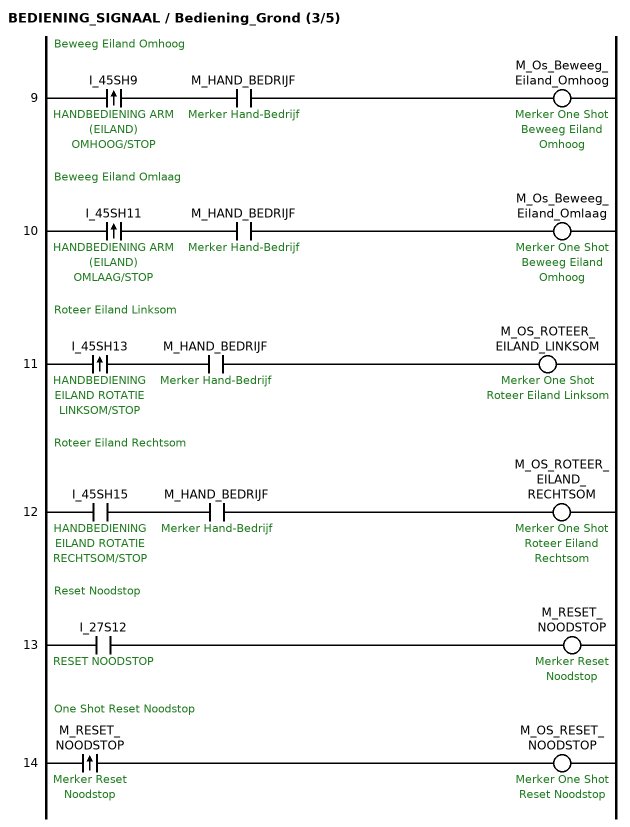
; [picture p96: BEDIENING_SIGNAAL / Bediening_Grond, rungs 9-14]
; rung 9: Beweeg Eiland Omhoog
@LD I_45SH9  ; HANDBEDIENING ARM (EILAND) OMHOOG/STOP
AND M_HAND_BEDRIJF  ; Merker Hand-Bedrijf
OUT M_Os_Beweeg_Eiland_Omhoog  ; Merker One Shot Beweeg Eiland Omhoog
; rung 10: Beweeg Eiland Omlaag
@LD I_45SH11  ; HANDBEDIENING ARM (EILAND) OMLAAG/STOP
AND M_HAND_BEDRIJF  ; Merker Hand-Bedrijf
OUT M_Os_Beweeg_Eiland_Omlaag  ; Merker One Shot Beweeg Eiland Omhoog
; rung 11: Roteer Eiland Linksom
@LD I_45SH13  ; HANDBEDIENING EILAND ROTATIE LINKSOM/STOP
AND M_HAND_BEDRIJF  ; Merker Hand-Bedrijf
OUT M_OS_ROTEER_EILAND_LINKSOM  ; Merker One Shot Roteer Eiland Linksom
; rung 12: Roteer Eiland Rechtsom
LD I_45SH15  ; HANDBEDIENING EILAND ROTATIE RECHTSOM/STOP
AND M_HAND_BEDRIJF  ; Merker Hand-Bedrijf
OUT M_OS_ROTEER_EILAND_RECHTSOM  ; Merker One Shot Roteer Eiland Rechtsom
; rung 13: Reset Noodstop
LD I_27S12  ; RESET NOODSTOP
OUT M_RESET_NOODSTOP  ; Merker Reset Noodstop
; rung 14: One Shot Reset Noodstop
@LD M_RESET_NOODSTOP  ; Merker Reset Noodstop
OUT M_OS_RESET_NOODSTOP  ; Merker One Shot  Reset Noodstop

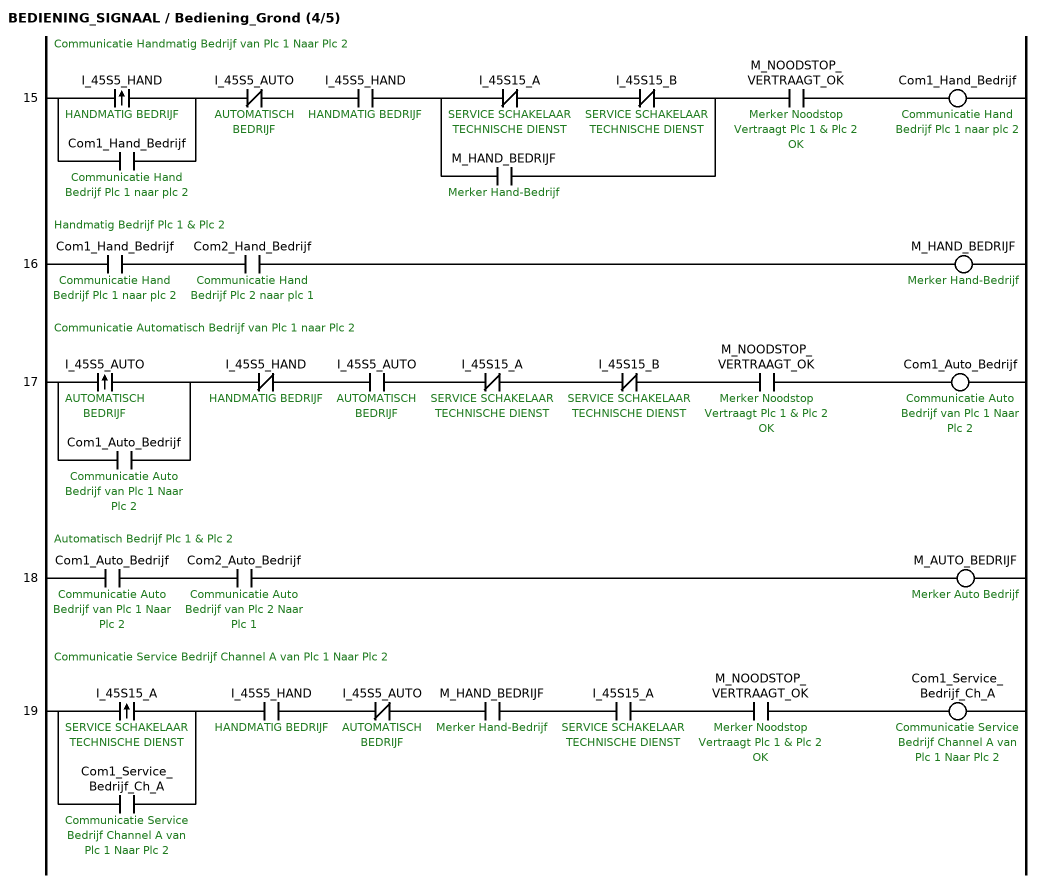
; rung 15: Communicatie Handmatig Bedrijf van Plc 1 Naar Plc 2
@LD I_45S5_HAND  ; HANDMATIG BEDRIJF
OR Com1_Hand_Bedrijf  ; Communicatie Hand Bedrijf Plc 1 naar plc 2
ANDNOT I_45S5_AUTO  ; AUTOMATISCH BEDRIJF
AND I_45S5_HAND  ; HANDMATIG BEDRIJF
LDNOT I_45S15_A  ; SERVICE SCHAKELAAR TECHNISCHE DIENST
ANDNOT I_45S15_B  ; SERVICE SCHAKELAAR TECHNISCHE DIENST
OR M_HAND_BEDRIJF  ; Merker Hand-Bedrijf
ANDLD
AND M_NOODSTOP_VERTRAAGT_OK  ; Merker Noodstop Vertraagt Plc 1 & Plc 2 OK
OUT Com1_Hand_Bedrijf  ; Communicatie Hand Bedrijf Plc 1 naar plc 2
; rung 16: Handmatig Bedrijf Plc 1 & Plc 2
LD Com1_Hand_Bedrijf  ; Communicatie Hand Bedrijf Plc 1 naar plc 2
AND Com2_Hand_Bedrijf  ; Communicatie Hand Bedrijf Plc 2 naar plc 1
OUT M_HAND_BEDRIJF  ; Merker Hand-Bedrijf
; rung 17: Communicatie Automatisch Bedrijf van Plc 1 naar Plc 2
@LD I_45S5_AUTO  ; AUTOMATISCH BEDRIJF
OR Com1_Auto_Bedrijf  ; Communicatie Auto Bedrijf van Plc 1 Naar Plc 2
ANDNOT I_45S5_HAND  ; HANDMATIG BEDRIJF
AND I_45S5_AUTO  ; AUTOMATISCH BEDRIJF
ANDNOT I_45S15_A  ; SERVICE SCHAKELAAR TECHNISCHE DIENST
ANDNOT I_45S15_B  ; SERVICE SCHAKELAAR TECHNISCHE DIENST
AND M_NOODSTOP_VERTRAAGT_OK  ; Merker Noodstop Vertraagt Plc 1 & Plc 2 OK
OUT Com1_Auto_Bedrijf  ; Communicatie Auto Bedrijf van Plc 1 Naar Plc 2
; rung 18: Automatisch Bedrijf Plc 1 & Plc 2
LD Com1_Auto_Bedrijf  ; Communicatie Auto Bedrijf van Plc 1 Naar Plc 2
AND Com2_Auto_Bedrijf  ; Communicatie Auto Bedrijf van Plc 2 Naar Plc 1
OUT M_AUTO_BEDRIJF  ; Merker Auto Bedrijf
; rung 19: Communicatie Service Bedrijf Channel A van Plc 1 Naar Plc 2
@LD I_45S15_A  ; SERVICE SCHAKELAAR TECHNISCHE DIENST
OR Com1_Service_Bedrijf_Ch_A  ; Communicatie Service Bedrijf Channel A van Plc 1 Naar Plc 2
AND I_45S5_HAND  ; HANDMATIG BEDRIJF
ANDNOT I_45S5_AUTO  ; AUTOMATISCH BEDRIJF
AND M_HAND_BEDRIJF  ; Merker Hand-Bedrijf
AND I_45S15_A  ; SERVICE SCHAKELAAR TECHNISCHE DIENST
AND M_NOODSTOP_VERTRAAGT_OK  ; Merker Noodstop Vertraagt Plc 1 & Plc 2 OK
OUT Com1_Service_Bedrijf_Ch_A  ; Communicatie Service Bedrijf Channel A van Plc 1 Naar Plc 2

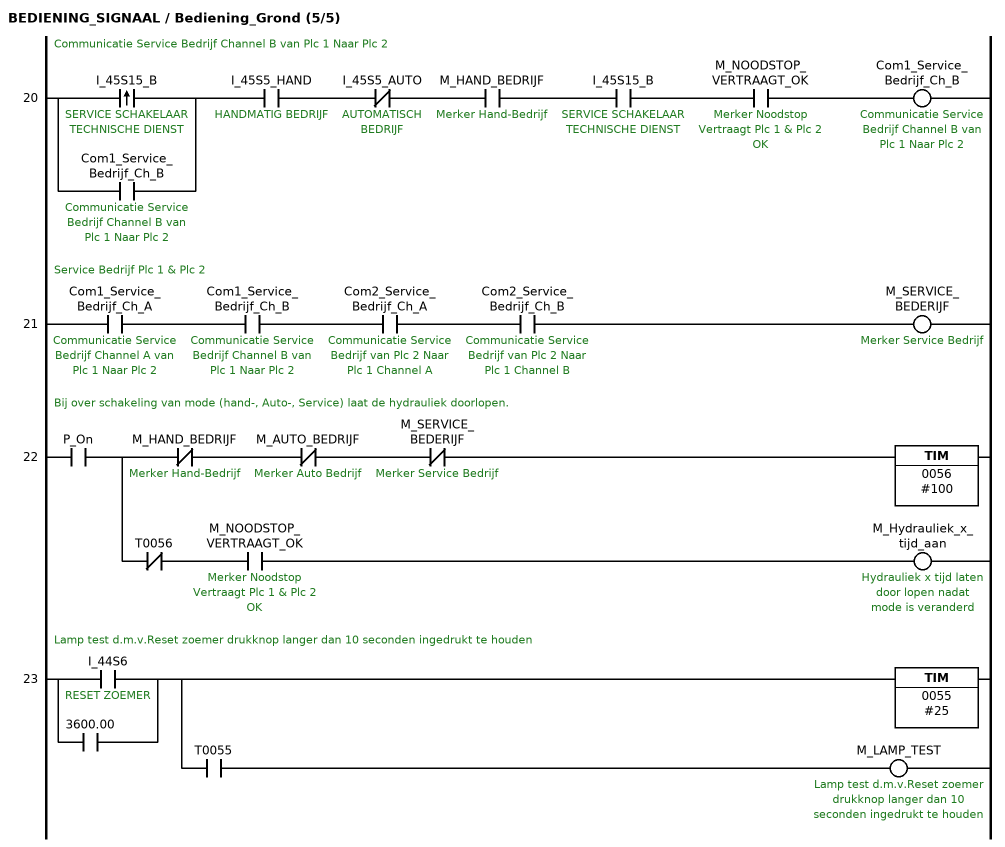
; rung 20: Communicatie Service Bedrijf Channel B van Plc 1 Naar Plc 2
@LD I_45S15_B  ; SERVICE SCHAKELAAR TECHNISCHE DIENST
OR Com1_Service_Bedrijf_Ch_B  ; Communicatie Service Bedrijf Channel B van Plc 1 Naar Plc 2
AND I_45S5_HAND  ; HANDMATIG BEDRIJF
ANDNOT I_45S5_AUTO  ; AUTOMATISCH BEDRIJF
AND M_HAND_BEDRIJF  ; Merker Hand-Bedrijf
AND I_45S15_B  ; SERVICE SCHAKELAAR TECHNISCHE DIENST
AND M_NOODSTOP_VERTRAAGT_OK  ; Merker Noodstop Vertraagt Plc 1 & Plc 2 OK
OUT Com1_Service_Bedrijf_Ch_B  ; Communicatie Service Bedrijf Channel B van Plc 1 Naar Plc 2
; rung 21: Service Bedrijf Plc 1 & Plc 2
LD Com1_Service_Bedrijf_Ch_A  ; Communicatie Service Bedrijf Channel A van Plc 1 Naar Plc 2
AND Com1_Service_Bedrijf_Ch_B  ; Communicatie Service Bedrijf Channel B van Plc 1 Naar Plc 2
AND Com2_Service_Bedrijf_Ch_A  ; Communicatie Service Bedrijf van Plc 2 Naar Plc 1 Channel A
AND Com2_Service_Bedrijf_Ch_B  ; Communicatie Service Bedrijf van Plc 2 Naar Plc 1 Channel B
OUT M_SERVICE_BEDERIJF  ; Merker Service Bedrijf
; rung 22: Bij over schakeling van mode (hand-, Auto-, Service) laat de hydrauliek doorlopen.
LD P_On
OUT TR0
ANDNOT M_HAND_BEDRIJF  ; Merker Hand-Bedrijf
ANDNOT M_AUTO_BEDRIJF  ; Merker Auto Bedrijf
ANDNOT M_SERVICE_BEDERIJF  ; Merker Service Bedrijf
TIM 0056 #100
LD TR0
ANDNOT T0056
AND M_NOODSTOP_VERTRAAGT_OK  ; Merker Noodstop Vertraagt Plc 1 & Plc 2 OK
OUT M_Hydrauliek_x_tijd_aan  ; Hydrauliek x tijd laten door lopen nadat mode is veranderd
; rung 23: Lamp test d.m.v.Reset zoemer drukknop langer dan 10 seconden ingedrukt te houden
LD I_44S6  ; RESET ZOEMER
OR 3600.00
TIM 0055 #25
AND T0055
OUT M_LAMP_TEST  ; Lamp test d.m.v.Reset zoemer drukknop langer dan 10 seconden ingedrukt te houden

### Section Sinalering_Grond

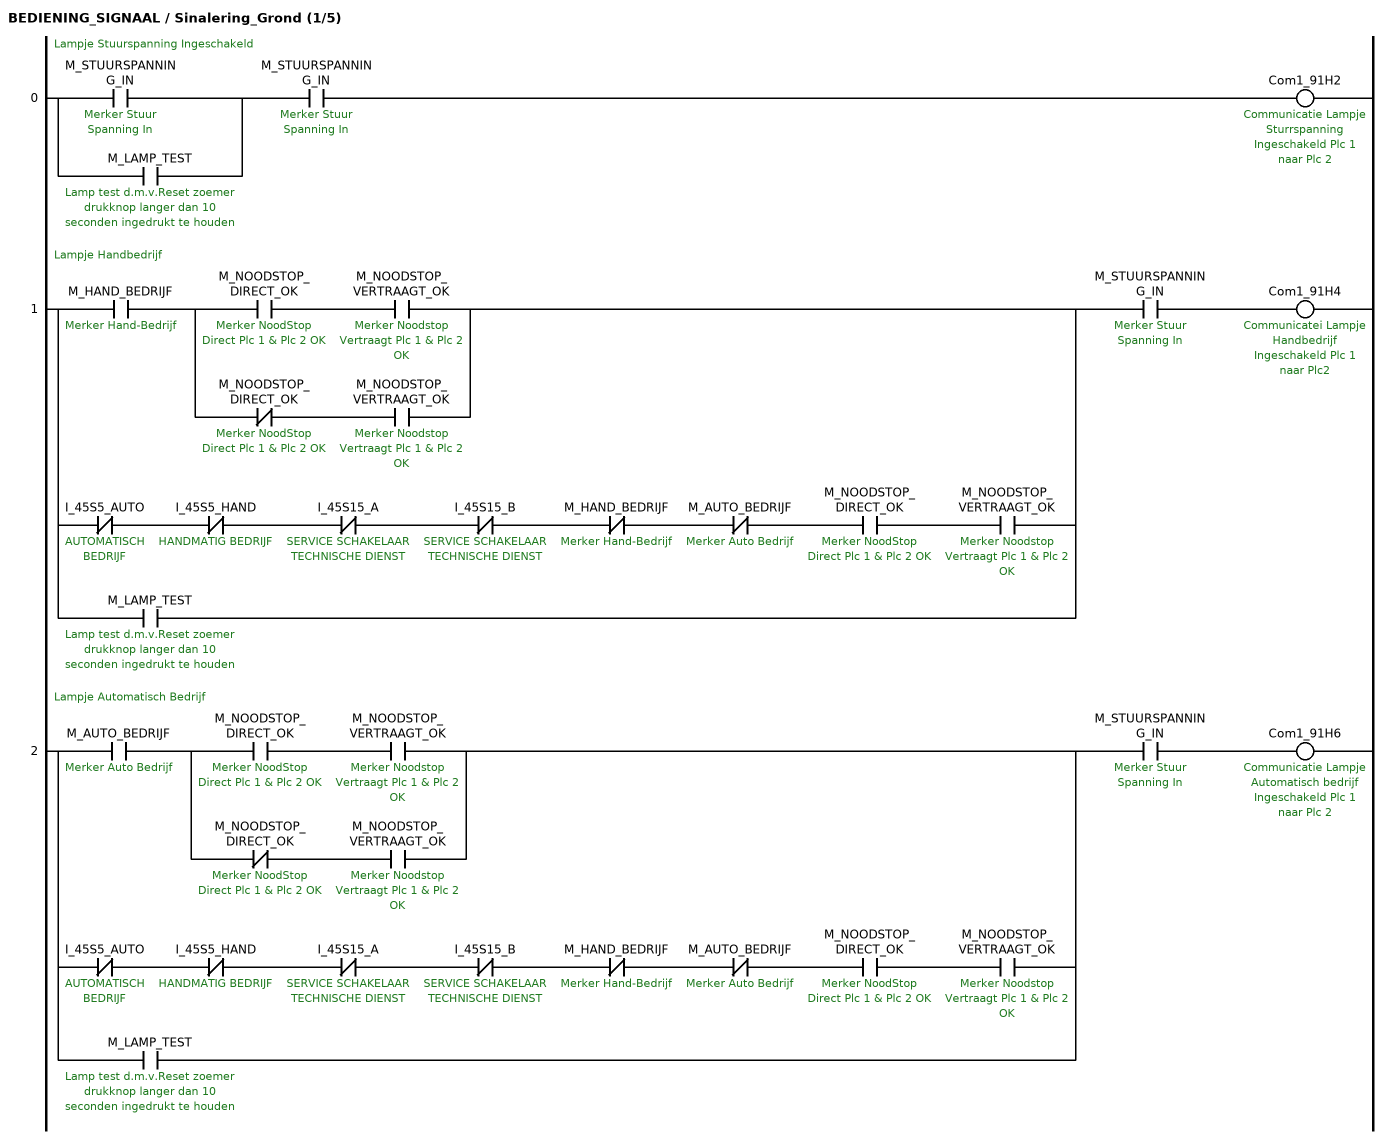
; rung 0: Lampje Stuurspanning Ingeschakeld
LD M_STUURSPANNING_IN  ; Merker Stuur Spanning In
OR M_LAMP_TEST  ; Lamp test d.m.v.Reset zoemer drukknop langer dan 10 seconden ingedrukt te houden
AND M_STUURSPANNING_IN  ; Merker Stuur Spanning In
OUT Com1_91H2  ; Communicatie Lampje Sturrspanning Ingeschakeld Plc 1 naar Plc 2
; rung 1: Lampje Handbedrijf
LD M_HAND_BEDRIJF  ; Merker Hand-Bedrijf
LD M_NOODSTOP_DIRECT_OK  ; Merker NoodStop Direct Plc 1 & Plc 2 OK
AND M_NOODSTOP_VERTRAAGT_OK  ; Merker Noodstop Vertraagt Plc 1 & Plc 2 OK
LDNOT M_NOODSTOP_DIRECT_OK  ; Merker NoodStop Direct Plc 1 & Plc 2 OK
AND M_NOODSTOP_VERTRAAGT_OK  ; Merker Noodstop Vertraagt Plc 1 & Plc 2 OK
ORLD
ANDLD
LDNOT I_45S5_AUTO  ; AUTOMATISCH BEDRIJF
ANDNOT I_45S5_HAND  ; HANDMATIG BEDRIJF
ANDNOT I_45S15_A  ; SERVICE SCHAKELAAR TECHNISCHE DIENST
ANDNOT I_45S15_B  ; SERVICE SCHAKELAAR TECHNISCHE DIENST
ANDNOT M_HAND_BEDRIJF  ; Merker Hand-Bedrijf
ANDNOT M_AUTO_BEDRIJF  ; Merker Auto Bedrijf
AND M_NOODSTOP_DIRECT_OK  ; Merker NoodStop Direct Plc 1 & Plc 2 OK
AND M_NOODSTOP_VERTRAAGT_OK  ; Merker Noodstop Vertraagt Plc 1 & Plc 2 OK
ORLD
OR M_LAMP_TEST  ; Lamp test d.m.v.Reset zoemer drukknop langer dan 10 seconden ingedrukt te houden
AND M_STUURSPANNING_IN  ; Merker Stuur Spanning In
OUT Com1_91H4  ; Communicatei Lampje Handbedrijf Ingeschakeld Plc 1 naar Plc2
; rung 2: Lampje Automatisch Bedrijf
LD M_AUTO_BEDRIJF  ; Merker Auto Bedrijf
LD M_NOODSTOP_DIRECT_OK  ; Merker NoodStop Direct Plc 1 & Plc 2 OK
AND M_NOODSTOP_VERTRAAGT_OK  ; Merker Noodstop Vertraagt Plc 1 & Plc 2 OK
LDNOT M_NOODSTOP_DIRECT_OK  ; Merker NoodStop Direct Plc 1 & Plc 2 OK
AND M_NOODSTOP_VERTRAAGT_OK  ; Merker Noodstop Vertraagt Plc 1 & Plc 2 OK
ORLD
ANDLD
LDNOT I_45S5_AUTO  ; AUTOMATISCH BEDRIJF
ANDNOT I_45S5_HAND  ; HANDMATIG BEDRIJF
ANDNOT I_45S15_A  ; SERVICE SCHAKELAAR TECHNISCHE DIENST
ANDNOT I_45S15_B  ; SERVICE SCHAKELAAR TECHNISCHE DIENST
ANDNOT M_HAND_BEDRIJF  ; Merker Hand-Bedrijf
ANDNOT M_AUTO_BEDRIJF  ; Merker Auto Bedrijf
AND M_NOODSTOP_DIRECT_OK  ; Merker NoodStop Direct Plc 1 & Plc 2 OK
AND M_NOODSTOP_VERTRAAGT_OK  ; Merker Noodstop Vertraagt Plc 1 & Plc 2 OK
ORLD
OR M_LAMP_TEST  ; Lamp test d.m.v.Reset zoemer drukknop langer dan 10 seconden ingedrukt te houden
AND M_STUURSPANNING_IN  ; Merker Stuur Spanning In
OUT Com1_91H6  ; Communicatie Lampje Automatisch bedrijf Ingeschakeld Plc 1 naar Plc 2

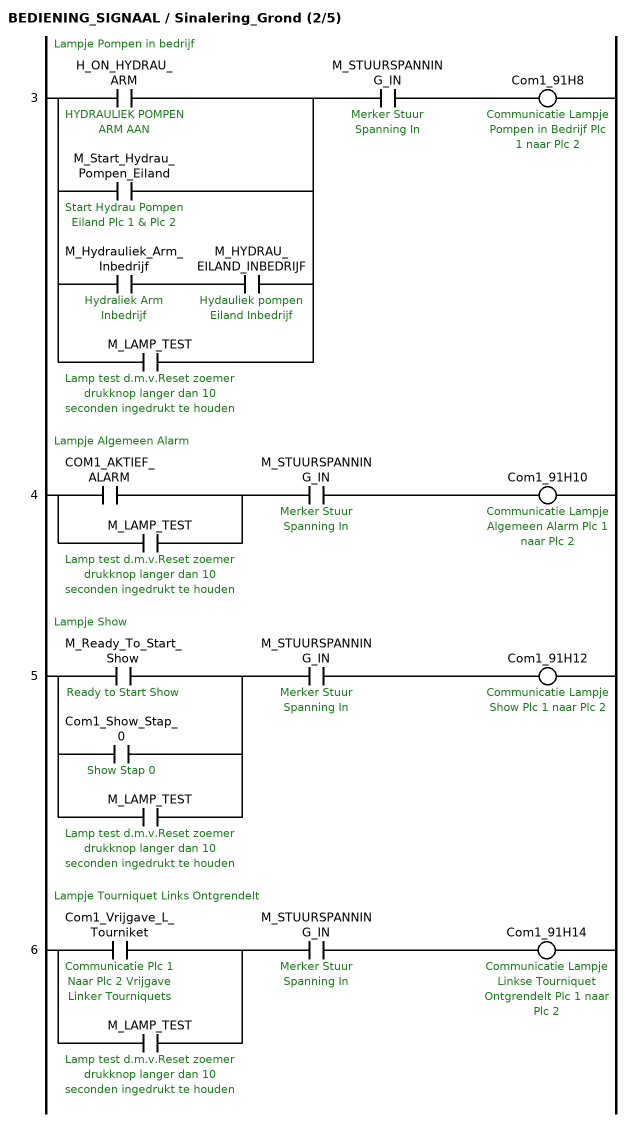
; rung 3: Lampje Pompen in bedrijf
LD H_ON_HYDRAU_ARM  ; HYDRAULIEK POMPEN ARM AAN
OR M_Start_Hydrau_Pompen_Eiland  ; Start Hydrau Pompen Eiland Plc 1 & Plc 2
LD M_Hydrauliek_Arm_Inbedrijf  ; Hydraliek Arm Inbedrijf
AND M_HYDRAU_EILAND_INBEDRIJF  ; Hydauliek pompen Eiland Inbedrijf
ORLD
OR M_LAMP_TEST  ; Lamp test d.m.v.Reset zoemer drukknop langer dan 10 seconden ingedrukt te houden
AND M_STUURSPANNING_IN  ; Merker Stuur Spanning In
OUT Com1_91H8  ; Communicatie Lampje Pompen in Bedrijf Plc 1 naar Plc 2
; rung 4: Lampje Algemeen Alarm
LD COM1_AKTIEF_ALARM
OR M_LAMP_TEST  ; Lamp test d.m.v.Reset zoemer drukknop langer dan 10 seconden ingedrukt te houden
AND M_STUURSPANNING_IN  ; Merker Stuur Spanning In
OUT Com1_91H10  ; Communicatie Lampje Algemeen Alarm Plc 1 naar Plc 2
; rung 5: Lampje Show
LD M_Ready_To_Start_Show  ; Ready to Start Show
OR Com1_Show_Stap_0  ; Show Stap 0
OR M_LAMP_TEST  ; Lamp test d.m.v.Reset zoemer drukknop langer dan 10 seconden ingedrukt te houden
AND M_STUURSPANNING_IN  ; Merker Stuur Spanning In
OUT Com1_91H12  ; Communicatie Lampje Show Plc 1 naar Plc 2
; rung 6: Lampje Tourniquet Links Ontgrendelt
LD Com1_Vrijgave_L_Tourniket  ; Communicatie Plc 1 Naar Plc 2 Vrijgave Linker Tourniquets
OR M_LAMP_TEST  ; Lamp test d.m.v.Reset zoemer drukknop langer dan 10 seconden ingedrukt te houden
AND M_STUURSPANNING_IN  ; Merker Stuur Spanning In
OUT Com1_91H14  ; Communicatie Lampje Linkse Tourniquet Ontgrendelt Plc 1 naar Plc 2

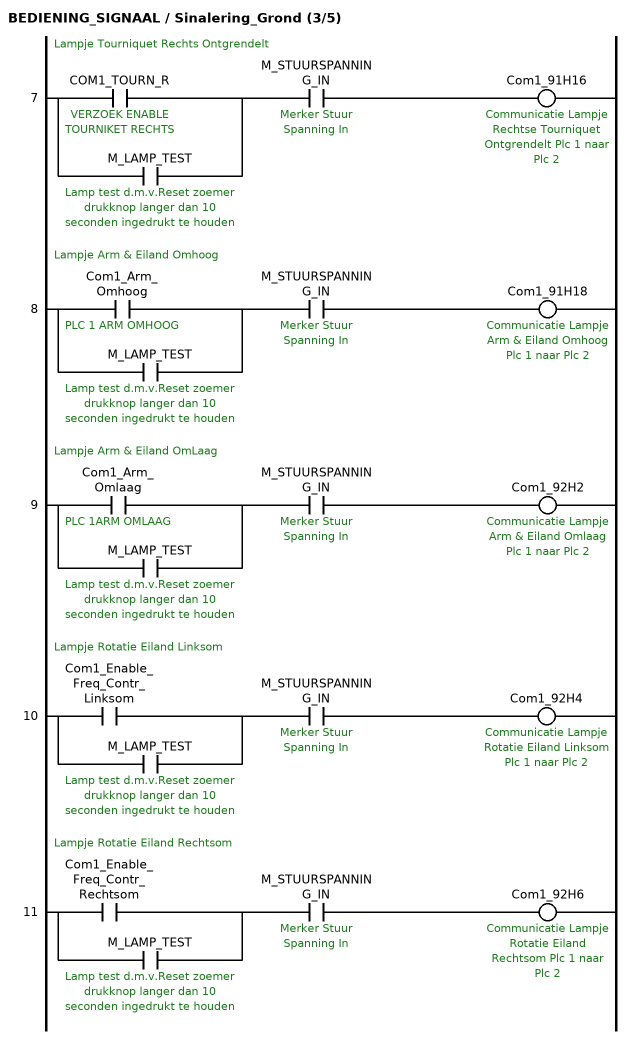
; rung 7: Lampje Tourniquet Rechts Ontgrendelt
LD COM1_TOURN_R  ; VERZOEK ENABLE TOURNIKET RECHTS
OR M_LAMP_TEST  ; Lamp test d.m.v.Reset zoemer drukknop langer dan 10 seconden ingedrukt te houden
AND M_STUURSPANNING_IN  ; Merker Stuur Spanning In
OUT Com1_91H16  ; Communicatie Lampje Rechtse Tourniquet Ontgrendelt Plc 1 naar Plc 2
; rung 8: Lampje Arm & Eiland Omhoog
LD Com1_Arm_Omhoog  ; PLC 1 ARM OMHOOG
OR M_LAMP_TEST  ; Lamp test d.m.v.Reset zoemer drukknop langer dan 10 seconden ingedrukt te houden
AND M_STUURSPANNING_IN  ; Merker Stuur Spanning In
OUT Com1_91H18  ; Communicatie Lampje Arm & Eiland Omhoog Plc 1 naar Plc 2
; rung 9: Lampje Arm & Eiland OmLaag
LD Com1_Arm_Omlaag  ; PLC 1ARM OMLAAG
OR M_LAMP_TEST  ; Lamp test d.m.v.Reset zoemer drukknop langer dan 10 seconden ingedrukt te houden
AND M_STUURSPANNING_IN  ; Merker Stuur Spanning In
OUT Com1_92H2  ; Communicatie Lampje Arm & Eiland Omlaag Plc 1 naar Plc 2
; rung 10: Lampje Rotatie Eiland Linksom
LD Com1_Enable_Freq_Contr_Linksom
OR M_LAMP_TEST  ; Lamp test d.m.v.Reset zoemer drukknop langer dan 10 seconden ingedrukt te houden
AND M_STUURSPANNING_IN  ; Merker Stuur Spanning In
OUT Com1_92H4  ; Communicatie Lampje Rotatie Eiland Linksom Plc 1 naar Plc 2
; rung 11: Lampje Rotatie Eiland Rechtsom
LD Com1_Enable_Freq_Contr_Rechtsom
OR M_LAMP_TEST  ; Lamp test d.m.v.Reset zoemer drukknop langer dan 10 seconden ingedrukt te houden
AND M_STUURSPANNING_IN  ; Merker Stuur Spanning In
OUT Com1_92H6  ; Communicatie Lampje Rotatie Eiland Rechtsom Plc 1 naar Plc 2

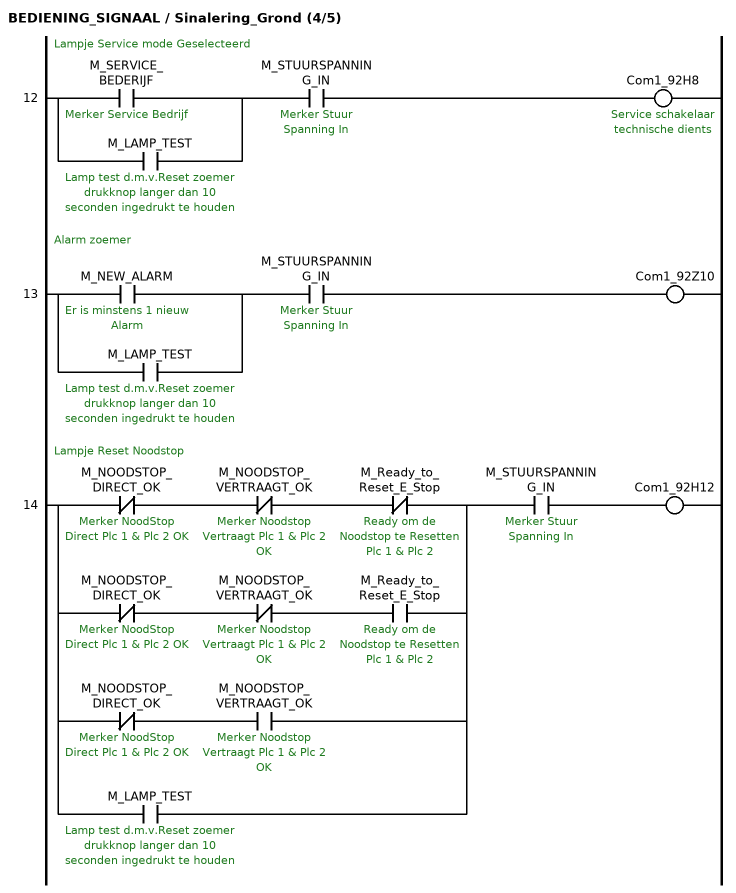
; rung 12: Lampje Service mode Geselecteerd
LD M_SERVICE_BEDERIJF  ; Merker Service Bedrijf
OR M_LAMP_TEST  ; Lamp test d.m.v.Reset zoemer drukknop langer dan 10 seconden ingedrukt te houden
AND M_STUURSPANNING_IN  ; Merker Stuur Spanning In
OUT Com1_92H8  ; Service schakelaar technische dients
; rung 13: Alarm zoemer
LD M_NEW_ALARM  ; Er is minstens 1 nieuw Alarm
OR M_LAMP_TEST  ; Lamp test d.m.v.Reset zoemer drukknop langer dan 10 seconden ingedrukt te houden
AND M_STUURSPANNING_IN  ; Merker Stuur Spanning In
OUT Com1_92Z10
; rung 14: Lampje Reset Noodstop
LDNOT M_NOODSTOP_DIRECT_OK  ; Merker NoodStop Direct Plc 1 & Plc 2 OK
ANDNOT M_NOODSTOP_VERTRAAGT_OK  ; Merker Noodstop Vertraagt Plc 1 & Plc 2 OK
ANDNOT M_Ready_to_Reset_E_Stop  ; Ready om de Noodstop te Resetten Plc 1 & Plc 2
LDNOT M_NOODSTOP_DIRECT_OK  ; Merker NoodStop Direct Plc 1 & Plc 2 OK
ANDNOT M_NOODSTOP_VERTRAAGT_OK  ; Merker Noodstop Vertraagt Plc 1 & Plc 2 OK
AND M_Ready_to_Reset_E_Stop  ; Ready om de Noodstop te Resetten Plc 1 & Plc 2
ORLD
LDNOT M_NOODSTOP_DIRECT_OK  ; Merker NoodStop Direct Plc 1 & Plc 2 OK
AND M_NOODSTOP_VERTRAAGT_OK  ; Merker Noodstop Vertraagt Plc 1 & Plc 2 OK
ORLD
OR M_LAMP_TEST  ; Lamp test d.m.v.Reset zoemer drukknop langer dan 10 seconden ingedrukt te houden
AND M_STUURSPANNING_IN  ; Merker Stuur Spanning In
OUT Com1_92H12

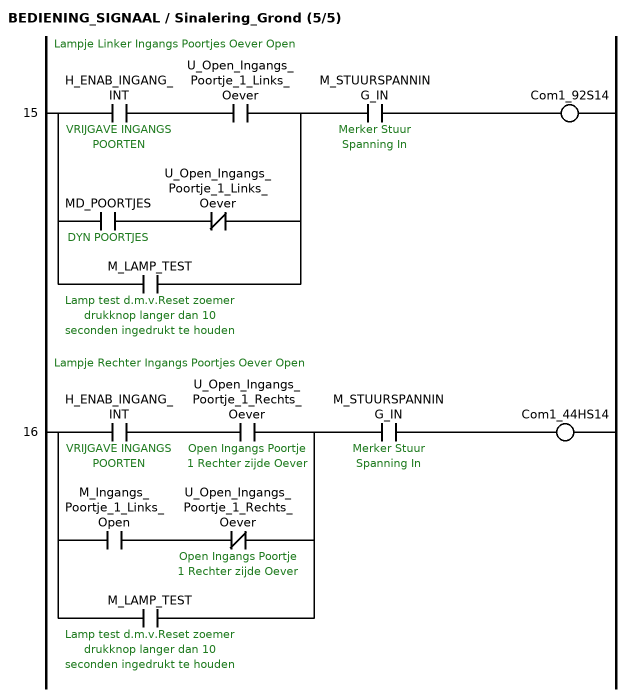
; rung 15: Lampje Linker Ingangs Poortjes Oever Open
LD H_ENAB_INGANG_INT  ; VRIJGAVE INGANGS POORTEN
AND U_Open_Ingangs_Poortje_1_Links_Oever
LD MD_POORTJES  ; DYN POORTJES
ANDNOT U_Open_Ingangs_Poortje_1_Links_Oever
ORLD
OR M_LAMP_TEST  ; Lamp test d.m.v.Reset zoemer drukknop langer dan 10 seconden ingedrukt te houden
AND M_STUURSPANNING_IN  ; Merker Stuur Spanning In
OUT Com1_92S14
; rung 16: Lampje Rechter Ingangs Poortjes Oever Open
LD H_ENAB_INGANG_INT  ; VRIJGAVE INGANGS POORTEN
AND U_Open_Ingangs_Poortje_1_Rechts_Oever  ; Open Ingangs Poortje 1 Rechter zijde Oever
LD M_Ingangs_Poortje_1_Links_Open
ANDNOT U_Open_Ingangs_Poortje_1_Rechts_Oever  ; Open Ingangs Poortje 1 Rechter zijde Oever
ORLD
OR M_LAMP_TEST  ; Lamp test d.m.v.Reset zoemer drukknop langer dan 10 seconden ingedrukt te houden
AND M_STUURSPANNING_IN  ; Merker Stuur Spanning In
OUT Com1_44HS14

### Section Bediening_Eiland

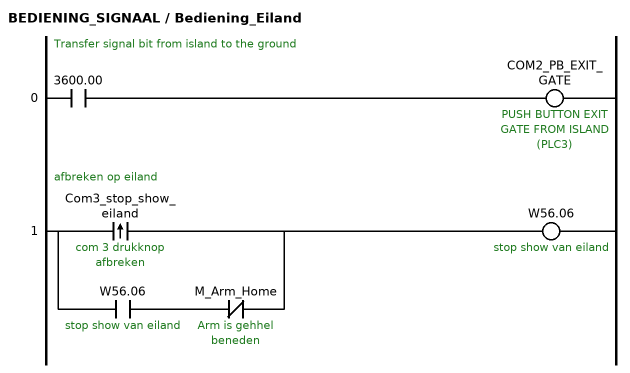
; rung 0: Transfer signal bit from island to the ground
LD 3600.00
OUT COM2_PB_EXIT_GATE  ; PUSH BUTTON EXIT GATE FROM ISLAND (PLC3)
; rung 1: afbreken op eiland
@LD Com3_stop_show_eiland  ; com 3 drukknop afbreken
LD W56.06  ; stop show van eiland
ANDNOT M_Arm_Home  ; Arm is gehhel beneden
ORLD
OUT W56.06  ; stop show van eiland

### Section Signalering_Eiland

### Section Bediening_Display_Eiland

### Section Signalering_Display_Eiland

### Section Einde_Bediening_Signalering
; rung 0
END(001)

## Program HOOFD_BESTURING (cyclic task 2)

### Section Afloop_Automatische_In_Uitgangs_Poortjes

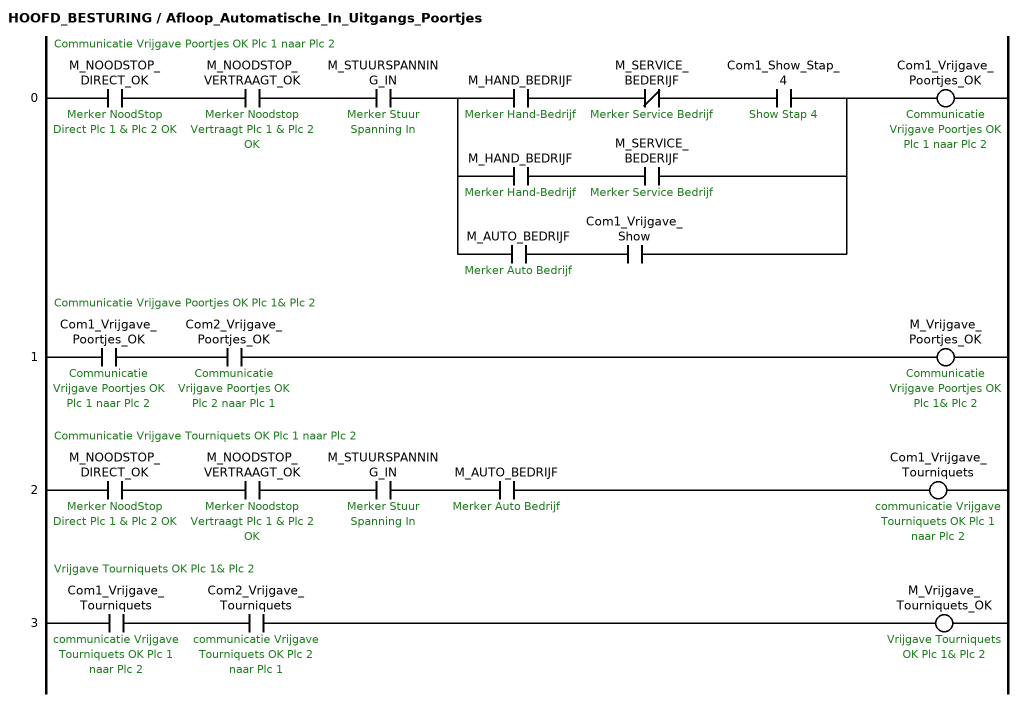
; rung 0: Communicatie Vrijgave Poortjes OK Plc 1 naar Plc 2
LD M_NOODSTOP_DIRECT_OK  ; Merker NoodStop Direct Plc 1 & Plc 2 OK
AND M_NOODSTOP_VERTRAAGT_OK  ; Merker Noodstop Vertraagt Plc 1 & Plc 2 OK
AND M_STUURSPANNING_IN  ; Merker Stuur Spanning In
LD M_HAND_BEDRIJF  ; Merker Hand-Bedrijf
ANDNOT M_SERVICE_BEDERIJF  ; Merker Service Bedrijf
AND Com1_Show_Stap_4  ; Show Stap 4
LD M_HAND_BEDRIJF  ; Merker Hand-Bedrijf
AND M_SERVICE_BEDERIJF  ; Merker Service Bedrijf
ORLD
LD M_AUTO_BEDRIJF  ; Merker Auto Bedrijf
AND Com1_Vrijgave_Show
ORLD
ANDLD
OUT Com1_Vrijgave_Poortjes_OK  ; Communicatie Vrijgave Poortjes OK Plc 1 naar Plc 2
; rung 1: Communicatie Vrijgave Poortjes OK Plc 1& Plc 2
LD Com1_Vrijgave_Poortjes_OK  ; Communicatie Vrijgave Poortjes OK Plc 1 naar Plc 2
AND Com2_Vrijgave_Poortjes_OK  ; Communicatie Vrijgave Poortjes OK Plc 2 naar Plc 1
OUT M_Vrijgave_Poortjes_OK  ; Communicatie Vrijgave Poortjes OK Plc 1& Plc 2
; rung 2: Communicatie Vrijgave Tourniquets OK Plc 1 naar Plc 2
LD M_NOODSTOP_DIRECT_OK  ; Merker NoodStop Direct Plc 1 & Plc 2 OK
AND M_NOODSTOP_VERTRAAGT_OK  ; Merker Noodstop Vertraagt Plc 1 & Plc 2 OK
AND M_STUURSPANNING_IN  ; Merker Stuur Spanning In
AND M_AUTO_BEDRIJF  ; Merker Auto Bedrijf
OUT Com1_Vrijgave_Tourniquets  ; communicatie Vrijgave Tourniquets OK Plc 1 naar Plc 2
; rung 3: Vrijgave Tourniquets OK Plc 1& Plc 2
LD Com1_Vrijgave_Tourniquets  ; communicatie Vrijgave Tourniquets OK Plc 1 naar Plc 2
AND Com2_Vrijgave_Tourniquets  ; communicatie Vrijgave Tourniquets OK Plc 2 naar Plc 1
OUT M_Vrijgave_Tourniquets_OK  ; Vrijgave Tourniquets OK Plc 1& Plc 2

### Section Afloop_Automatisch_Programma

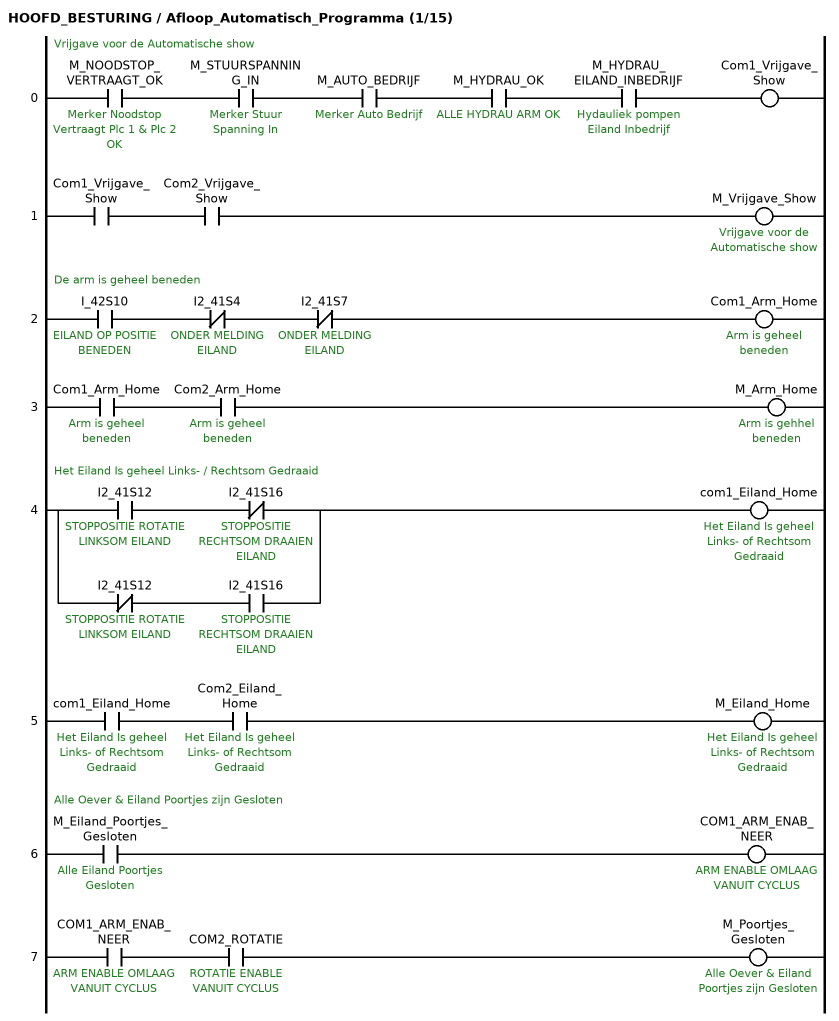
; rung 0: Vrijgave voor de Automatische show
LD M_NOODSTOP_VERTRAAGT_OK  ; Merker Noodstop Vertraagt Plc 1 & Plc 2 OK
AND M_STUURSPANNING_IN  ; Merker Stuur Spanning In
AND M_AUTO_BEDRIJF  ; Merker Auto Bedrijf
AND M_HYDRAU_OK  ; ALLE HYDRAU ARM OK
AND M_HYDRAU_EILAND_INBEDRIJF  ; Hydauliek pompen Eiland Inbedrijf
OUT Com1_Vrijgave_Show
; rung 1
LD Com1_Vrijgave_Show
AND Com2_Vrijgave_Show
OUT M_Vrijgave_Show  ; Vrijgave voor de Automatische show
; rung 2: De arm is geheel beneden
LD I_42S10  ; EILAND OP POSITIE BENEDEN
ANDNOT I2_41S4  ; ONDER MELDING EILAND
ANDNOT I2_41S7  ; ONDER MELDING EILAND
OUT Com1_Arm_Home  ; Arm is geheel beneden
; rung 3
LD Com1_Arm_Home  ; Arm is geheel beneden
AND Com2_Arm_Home  ; Arm is geheel beneden
OUT M_Arm_Home  ; Arm is gehhel beneden
; rung 4: Het Eiland Is geheel Links- / Rechtsom Gedraaid
LD I2_41S12  ; STOPPOSITIE ROTATIE LINKSOM EILAND
ANDNOT I2_41S16  ; STOPPOSITIE RECHTSOM DRAAIEN EILAND
LDNOT I2_41S12  ; STOPPOSITIE ROTATIE LINKSOM EILAND
AND I2_41S16  ; STOPPOSITIE RECHTSOM DRAAIEN EILAND
ORLD
OUT com1_Eiland_Home  ; Het Eiland Is geheel Links- of Rechtsom Gedraaid
; rung 5
LD com1_Eiland_Home  ; Het Eiland Is geheel Links- of Rechtsom Gedraaid
AND Com2_Eiland_Home  ; Het Eiland Is geheel Links- of Rechtsom Gedraaid
OUT M_Eiland_Home  ; Het Eiland Is geheel Links- of Rechtsom Gedraaid
; rung 6: Alle Oever & Eiland Poortjes zijn Gesloten
LD M_Eiland_Poortjes_Gesloten  ; Alle Eiland Poortjes Gesloten
OUT COM1_ARM_ENAB_NEER  ; ARM ENABLE OMLAAG  VANUIT CYCLUS
; rung 7
LD COM1_ARM_ENAB_NEER  ; ARM ENABLE OMLAAG  VANUIT CYCLUS
AND COM2_ROTATIE  ; ROTATIE ENABLE VANUIT CYCLUS
OUT M_Poortjes_Gesloten  ; Alle Oever & Eiland Poortjes zijn Gesloten

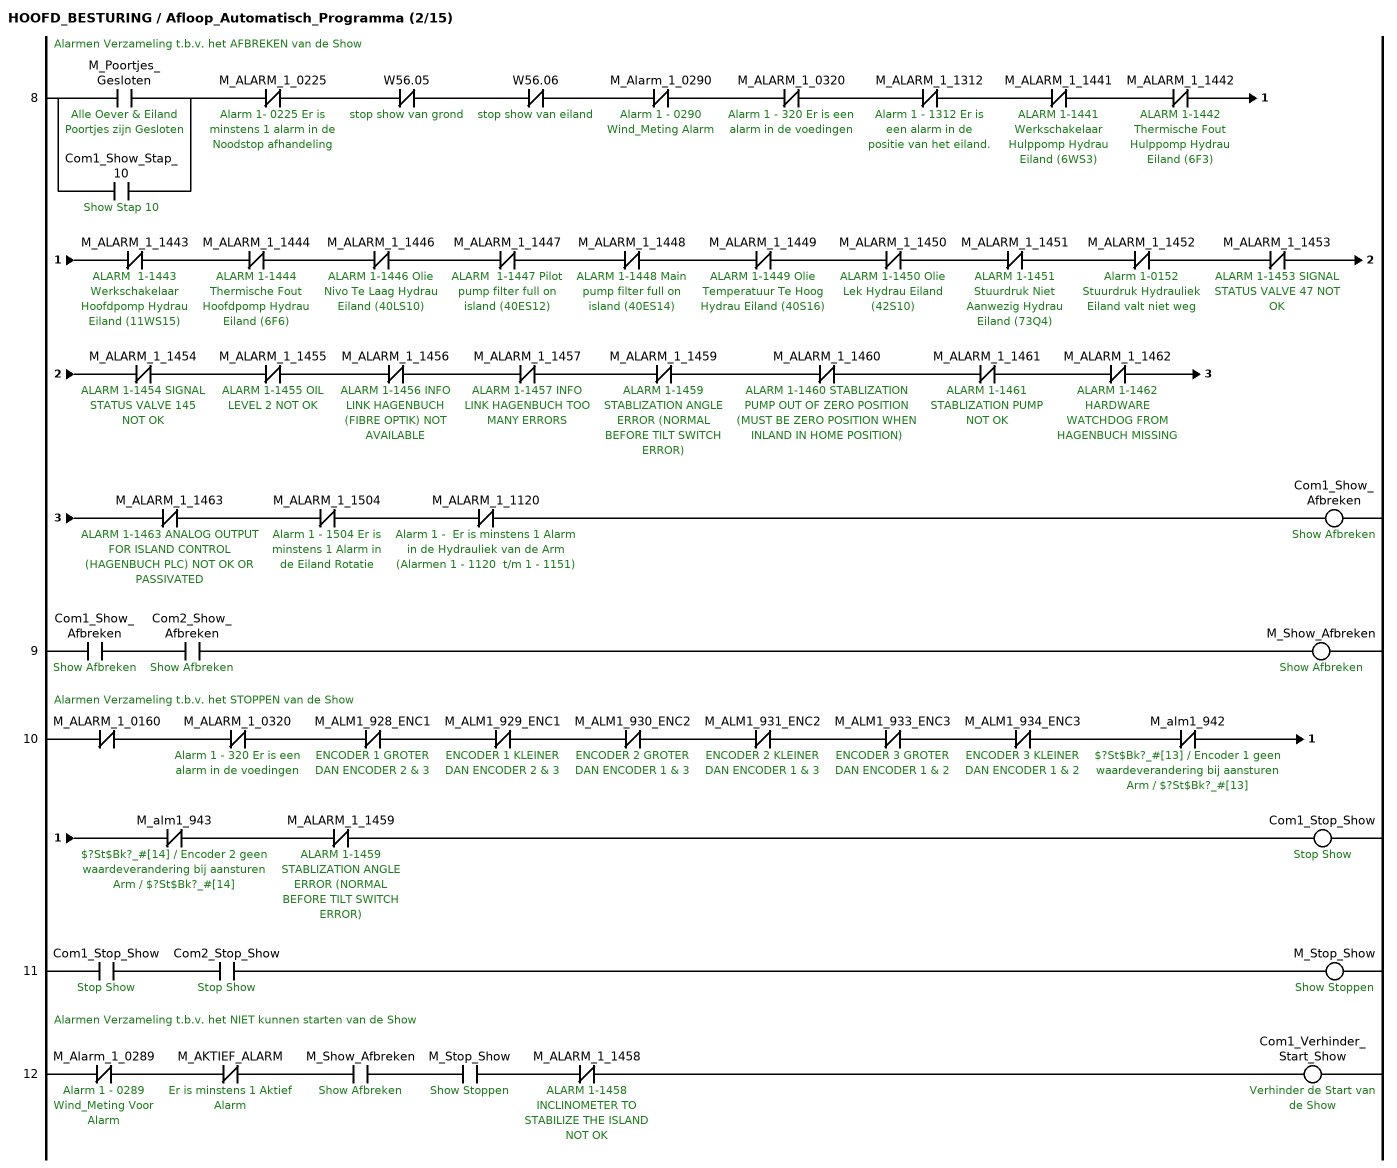
; rung 8: Alarmen Verzameling t.b.v. het AFBREKEN van de Show
LD M_Poortjes_Gesloten  ; Alle Oever & Eiland Poortjes zijn Gesloten
OR Com1_Show_Stap_10  ; Show Stap 10
ANDNOT M_ALARM_1_0225  ; Alarm 1- 0225 Er is minstens 1 alarm in de Noodstop afhandeling
ANDNOT W56.05  ; stop show van grond
ANDNOT W56.06  ; stop show van eiland
ANDNOT M_Alarm_1_0290  ; Alarm 1 - 0290 Wind_Meting Alarm
ANDNOT M_ALARM_1_0320  ; Alarm 1 - 320 Er is een alarm in de voedingen
ANDNOT M_ALARM_1_1312  ; Alarm 1 - 1312 Er is een alarm in de positie van het eiland.
ANDNOT M_ALARM_1_1441  ; ALARM 1-1441 Werkschakelaar Hulppomp Hydrau Eiland (6WS3)
ANDNOT M_ALARM_1_1442  ; ALARM 1-1442 Thermische Fout Hulppomp Hydrau Eiland (6F3)
ANDNOT M_ALARM_1_1443  ; ALARM  1-1443 Werkschakelaar Hoofdpomp Hydrau Eiland (11WS15)
ANDNOT M_ALARM_1_1444  ; ALARM 1-1444 Thermische Fout Hoofdpomp Hydrau Eiland (6F6)
ANDNOT M_ALARM_1_1446  ; ALARM 1-1446 Olie Nivo Te Laag Hydrau Eiland (40LS10)
ANDNOT M_ALARM_1_1447  ; ALARM  1-1447 Pilot pump filter full on island (40ES12)
ANDNOT M_ALARM_1_1448  ; ALARM 1-1448 Main pump filter full on island (40ES14)
ANDNOT M_ALARM_1_1449  ; ALARM 1-1449 Olie Temperatuur Te Hoog Hydrau Eiland (40S16)
ANDNOT M_ALARM_1_1450  ; ALARM 1-1450 Olie Lek Hydrau Eiland (42S10)
ANDNOT M_ALARM_1_1451  ; ALARM 1-1451 Stuurdruk Niet Aanwezig Hydrau Eiland (73Q4)
ANDNOT M_ALARM_1_1452  ; Alarm 1-0152 Stuurdruk Hydrauliek Eiland valt niet weg
ANDNOT M_ALARM_1_1453  ; ALARM 1-1453 SIGNAL STATUS VALVE 47 NOT OK
ANDNOT M_ALARM_1_1454  ; ALARM 1-1454 SIGNAL STATUS VALVE 145 NOT OK
ANDNOT M_ALARM_1_1455  ; ALARM 1-1455 OIL LEVEL 2 NOT OK
ANDNOT M_ALARM_1_1456  ; ALARM 1-1456 INFO LINK HAGENBUCH (FIBRE OPTIK) NOT AVAILABLE
ANDNOT M_ALARM_1_1457  ; ALARM 1-1457 INFO LINK HAGENBUCH TOO MANY ERRORS
ANDNOT M_ALARM_1_1459  ; ALARM 1-1459 STABLIZATION ANGLE ERROR (NORMAL BEFORE TILT SWITCH ERROR)
ANDNOT M_ALARM_1_1460  ; ALARM 1-1460 STABLIZATION PUMP OUT OF ZERO POSITION (MUST BE ZERO POSITION WHEN INLAND IN HOME POSITION)
ANDNOT M_ALARM_1_1461  ; ALARM 1-1461 STABLIZATION PUMP NOT OK
ANDNOT M_ALARM_1_1462  ; ALARM 1-1462 HARDWARE WATCHDOG FROM HAGENBUCH MISSING
ANDNOT M_ALARM_1_1463  ; ALARM 1-1463 ANALOG OUTPUT FOR ISLAND CONTROL (HAGENBUCH PLC) NOT OK OR PASSIVATED
ANDNOT M_ALARM_1_1504  ; Alarm 1 - 1504 Er is minstens 1 Alarm in de Eiland Rotatie
ANDNOT M_ALARM_1_1120  ; Alarm 1 -  Er is minstens 1 Alarm in de Hydrauliek van de Arm  (Alarmen 1 - 1120  t/m 1 - 1151)
OUT Com1_Show_Afbreken  ; Show Afbreken
; rung 9
LD Com1_Show_Afbreken  ; Show Afbreken
AND Com2_Show_Afbreken  ; Show Afbreken
OUT M_Show_Afbreken  ; Show Afbreken
; rung 10: Alarmen Verzameling t.b.v. het STOPPEN van de Show
LDNOT M_ALARM_1_0160
ANDNOT M_ALARM_1_0320  ; Alarm 1 - 320 Er is een alarm in de voedingen
ANDNOT M_ALM1_928_ENC1  ; ENCODER 1 GROTER DAN ENCODER 2 & 3
ANDNOT M_ALM1_929_ENC1  ; ENCODER 1 KLEINER DAN ENCODER 2 & 3
ANDNOT M_ALM1_930_ENC2  ; ENCODER 2 GROTER DAN ENCODER 1 & 3
ANDNOT M_ALM1_931_ENC2  ; ENCODER 2 KLEINER DAN ENCODER 1 & 3
ANDNOT M_ALM1_933_ENC3  ; ENCODER 3 GROTER DAN ENCODER 1 & 2
ANDNOT M_ALM1_934_ENC3  ; ENCODER 3 KLEINER DAN ENCODER 1 & 2
ANDNOT M_alm1_942  ; $?St$Bk?_#[13] / Encoder 1 geen waardeverandering bij aansturen Arm / $?St$Bk?_#[13]
ANDNOT M_alm1_943  ; $?St$Bk?_#[14] / Encoder 2 geen waardeverandering bij aansturen Arm / $?St$Bk?_#[14]
ANDNOT M_ALARM_1_1459  ; ALARM 1-1459 STABLIZATION ANGLE ERROR (NORMAL BEFORE TILT SWITCH ERROR)
OUT Com1_Stop_Show  ; Stop Show
; rung 11
LD Com1_Stop_Show  ; Stop Show
AND Com2_Stop_Show  ; Stop Show
OUT M_Stop_Show  ; Show Stoppen
; rung 12: Alarmen Verzameling t.b.v. het NIET kunnen starten van de Show
LDNOT M_Alarm_1_0289  ; Alarm 1 - 0289 Wind_Meting Voor Alarm
ANDNOT M_AKTIEF_ALARM  ; Er is minstens 1 Aktief Alarm
AND M_Show_Afbreken  ; Show Afbreken
AND M_Stop_Show  ; Show Stoppen
ANDNOT M_ALARM_1_1458  ; ALARM 1-1458 INCLINOMETER TO STABILIZE THE ISLAND NOT OK
OUT Com1_Verhinder_Start_Show  ; Verhinder de Start van de Show

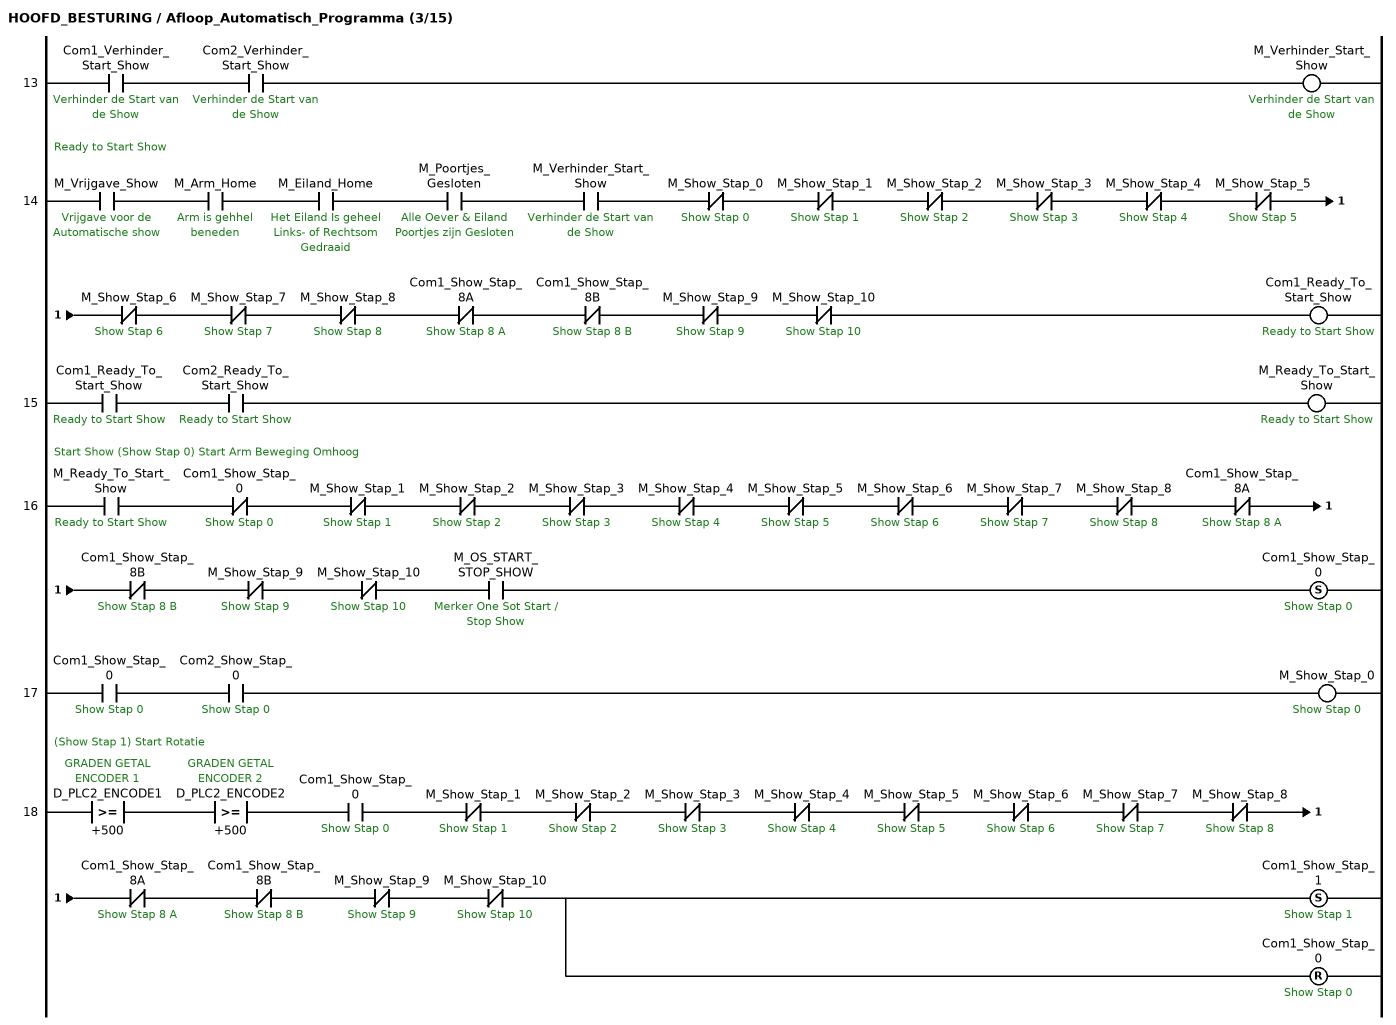
; rung 13
LD Com1_Verhinder_Start_Show  ; Verhinder de Start van de Show
AND Com2_Verhinder_Start_Show  ; Verhinder de Start van de Show
OUT M_Verhinder_Start_Show  ; Verhinder de Start van de Show
; rung 14: Ready to Start Show
LD M_Vrijgave_Show  ; Vrijgave voor de Automatische show
AND M_Arm_Home  ; Arm is gehhel beneden
AND M_Eiland_Home  ; Het Eiland Is geheel Links- of Rechtsom Gedraaid
AND M_Poortjes_Gesloten  ; Alle Oever & Eiland Poortjes zijn Gesloten
AND M_Verhinder_Start_Show  ; Verhinder de Start van de Show
ANDNOT M_Show_Stap_0  ; Show Stap 0
ANDNOT M_Show_Stap_1  ; Show Stap 1
ANDNOT M_Show_Stap_2  ; Show Stap 2
ANDNOT M_Show_Stap_3  ; Show Stap 3
ANDNOT M_Show_Stap_4  ; Show Stap 4
ANDNOT M_Show_Stap_5  ; Show Stap 5
ANDNOT M_Show_Stap_6  ; Show Stap 6
ANDNOT M_Show_Stap_7  ; Show Stap 7
ANDNOT M_Show_Stap_8  ; Show Stap 8
ANDNOT Com1_Show_Stap_8A  ; Show Stap 8 A
ANDNOT Com1_Show_Stap_8B  ; Show Stap 8 B
ANDNOT M_Show_Stap_9  ; Show Stap 9
ANDNOT M_Show_Stap_10  ; Show Stap 10
OUT Com1_Ready_To_Start_Show  ; Ready to Start Show
; rung 15
LD Com1_Ready_To_Start_Show  ; Ready to Start Show
AND Com2_Ready_To_Start_Show  ; Ready to Start Show
OUT M_Ready_To_Start_Show  ; Ready to Start Show
; rung 16: Start Show (Show Stap 0) Start Arm Beweging Omhoog
LD M_Ready_To_Start_Show  ; Ready to Start Show
ANDNOT Com1_Show_Stap_0  ; Show Stap 0
ANDNOT M_Show_Stap_1  ; Show Stap 1
ANDNOT M_Show_Stap_2  ; Show Stap 2
ANDNOT M_Show_Stap_3  ; Show Stap 3
ANDNOT M_Show_Stap_4  ; Show Stap 4
ANDNOT M_Show_Stap_5  ; Show Stap 5
ANDNOT M_Show_Stap_6  ; Show Stap 6
ANDNOT M_Show_Stap_7  ; Show Stap 7
ANDNOT M_Show_Stap_8  ; Show Stap 8
ANDNOT Com1_Show_Stap_8A  ; Show Stap 8 A
ANDNOT Com1_Show_Stap_8B  ; Show Stap 8 B
ANDNOT M_Show_Stap_9  ; Show Stap 9
ANDNOT M_Show_Stap_10  ; Show Stap 10
AND M_OS_START_STOP_SHOW  ; Merker One Sot Start / Stop Show
SET Com1_Show_Stap_0  ; Show Stap 0
; rung 17
LD Com1_Show_Stap_0  ; Show Stap 0
AND Com2_Show_Stap_0  ; Show Stap 0
OUT M_Show_Stap_0  ; Show Stap 0
; rung 18: (Show Stap 1) Start Rotatie
LD>=S(327) D_PLC2_ENCODE1 +500  ; GRADEN GETAL ENCODER 1
AND>=S(327) D_PLC2_ENCODE2 +500  ; GRADEN GETAL ENCODER 2
AND Com1_Show_Stap_0  ; Show Stap 0
ANDNOT M_Show_Stap_1  ; Show Stap 1
ANDNOT M_Show_Stap_2  ; Show Stap 2
ANDNOT M_Show_Stap_3  ; Show Stap 3
ANDNOT M_Show_Stap_4  ; Show Stap 4
ANDNOT M_Show_Stap_5  ; Show Stap 5
ANDNOT M_Show_Stap_6  ; Show Stap 6
ANDNOT M_Show_Stap_7  ; Show Stap 7
ANDNOT M_Show_Stap_8  ; Show Stap 8
ANDNOT Com1_Show_Stap_8A  ; Show Stap 8 A
ANDNOT Com1_Show_Stap_8B  ; Show Stap 8 B
ANDNOT M_Show_Stap_9  ; Show Stap 9
ANDNOT M_Show_Stap_10  ; Show Stap 10
SET Com1_Show_Stap_1  ; Show Stap 1
RSET Com1_Show_Stap_0  ; Show Stap 0

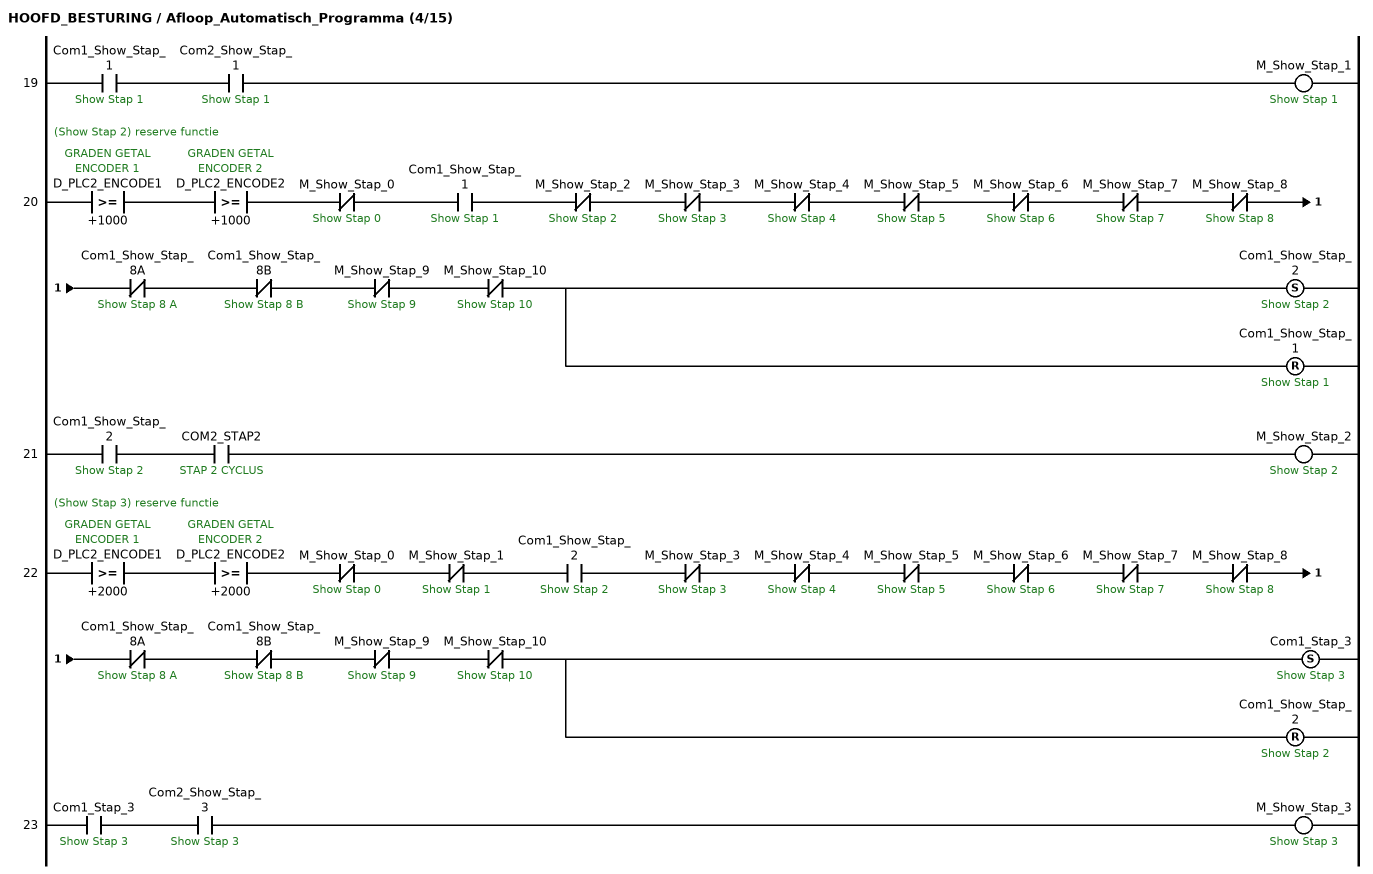
; rung 19
LD Com1_Show_Stap_1  ; Show Stap 1
AND Com2_Show_Stap_1  ; Show Stap 1
OUT M_Show_Stap_1  ; Show Stap 1
; rung 20: (Show Stap 2) reserve functie
LD>=S(327) D_PLC2_ENCODE1 +1000  ; GRADEN GETAL ENCODER 1
AND>=S(327) D_PLC2_ENCODE2 +1000  ; GRADEN GETAL ENCODER 2
ANDNOT M_Show_Stap_0  ; Show Stap 0
AND Com1_Show_Stap_1  ; Show Stap 1
ANDNOT M_Show_Stap_2  ; Show Stap 2
ANDNOT M_Show_Stap_3  ; Show Stap 3
ANDNOT M_Show_Stap_4  ; Show Stap 4
ANDNOT M_Show_Stap_5  ; Show Stap 5
ANDNOT M_Show_Stap_6  ; Show Stap 6
ANDNOT M_Show_Stap_7  ; Show Stap 7
ANDNOT M_Show_Stap_8  ; Show Stap 8
ANDNOT Com1_Show_Stap_8A  ; Show Stap 8 A
ANDNOT Com1_Show_Stap_8B  ; Show Stap 8 B
ANDNOT M_Show_Stap_9  ; Show Stap 9
ANDNOT M_Show_Stap_10  ; Show Stap 10
SET Com1_Show_Stap_2  ; Show Stap 2
RSET Com1_Show_Stap_1  ; Show Stap 1
; rung 21
LD Com1_Show_Stap_2  ; Show Stap 2
AND COM2_STAP2  ; STAP 2 CYCLUS
OUT M_Show_Stap_2  ; Show Stap 2
; rung 22: (Show Stap 3) reserve functie
LD>=S(327) D_PLC2_ENCODE1 +2000  ; GRADEN GETAL ENCODER 1
AND>=S(327) D_PLC2_ENCODE2 +2000  ; GRADEN GETAL ENCODER 2
ANDNOT M_Show_Stap_0  ; Show Stap 0
ANDNOT M_Show_Stap_1  ; Show Stap 1
AND Com1_Show_Stap_2  ; Show Stap 2
ANDNOT M_Show_Stap_3  ; Show Stap 3
ANDNOT M_Show_Stap_4  ; Show Stap 4
ANDNOT M_Show_Stap_5  ; Show Stap 5
ANDNOT M_Show_Stap_6  ; Show Stap 6
ANDNOT M_Show_Stap_7  ; Show Stap 7
ANDNOT M_Show_Stap_8  ; Show Stap 8
ANDNOT Com1_Show_Stap_8A  ; Show Stap 8 A
ANDNOT Com1_Show_Stap_8B  ; Show Stap 8 B
ANDNOT M_Show_Stap_9  ; Show Stap 9
ANDNOT M_Show_Stap_10  ; Show Stap 10
SET Com1_Stap_3  ; Show Stap 3
RSET Com1_Show_Stap_2  ; Show Stap 2
; rung 23
LD Com1_Stap_3  ; Show Stap 3
AND Com2_Show_Stap_3  ; Show Stap 3
OUT M_Show_Stap_3  ; Show Stap 3

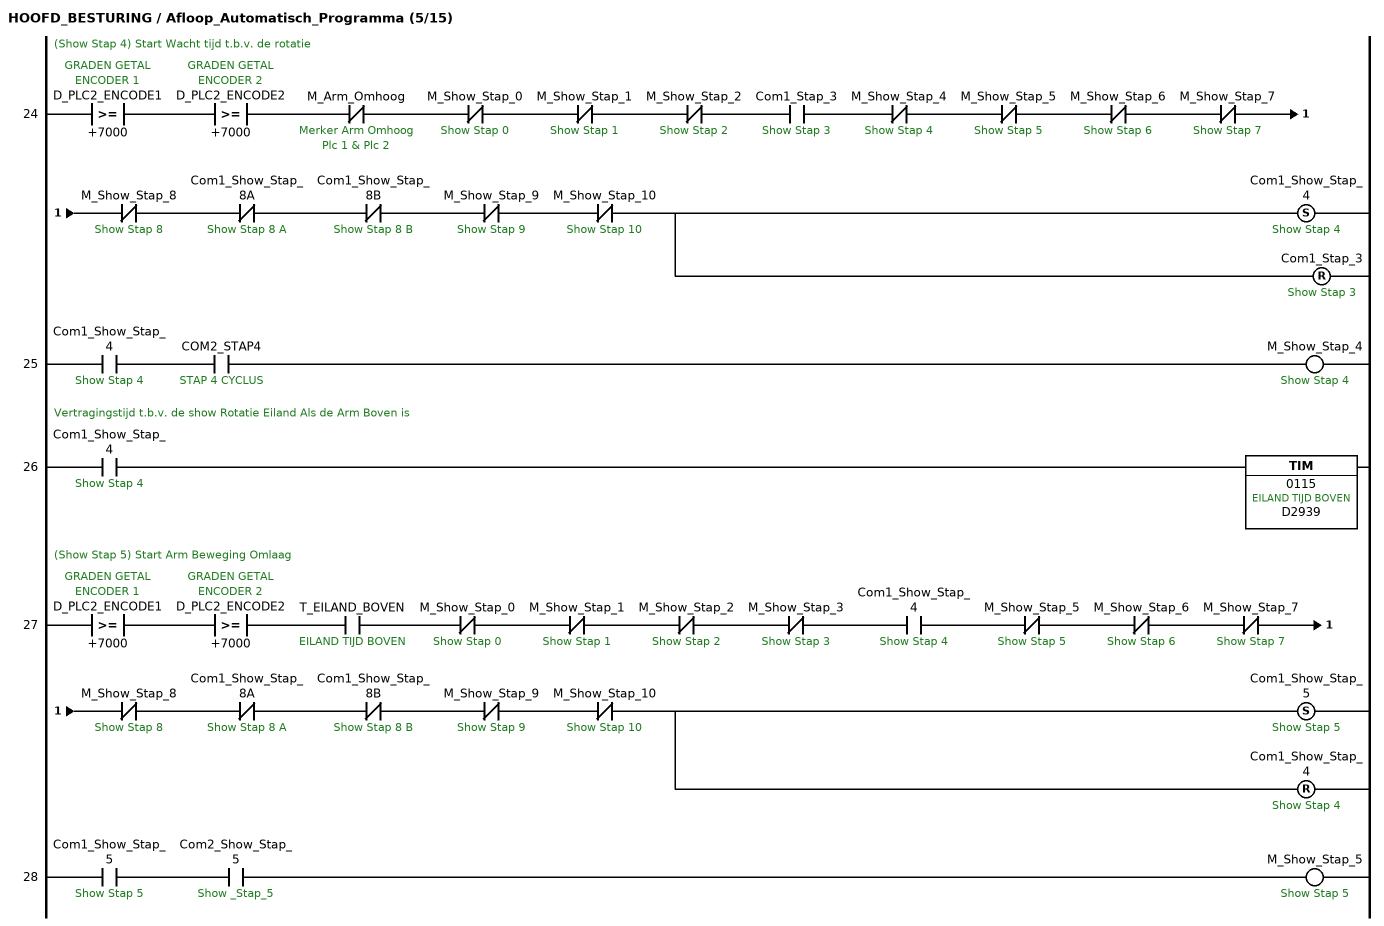
; rung 24: (Show Stap 4) Start Wacht tijd t.b.v. de rotatie
LD>=S(327) D_PLC2_ENCODE1 +7000  ; GRADEN GETAL ENCODER 1
AND>=S(327) D_PLC2_ENCODE2 +7000  ; GRADEN GETAL ENCODER 2
ANDNOT M_Arm_Omhoog  ; Merker Arm Omhoog Plc 1 & Plc 2
ANDNOT M_Show_Stap_0  ; Show Stap 0
ANDNOT M_Show_Stap_1  ; Show Stap 1
ANDNOT M_Show_Stap_2  ; Show Stap 2
AND Com1_Stap_3  ; Show Stap 3
ANDNOT M_Show_Stap_4  ; Show Stap 4
ANDNOT M_Show_Stap_5  ; Show Stap 5
ANDNOT M_Show_Stap_6  ; Show Stap 6
ANDNOT M_Show_Stap_7  ; Show Stap 7
ANDNOT M_Show_Stap_8  ; Show Stap 8
ANDNOT Com1_Show_Stap_8A  ; Show Stap 8 A
ANDNOT Com1_Show_Stap_8B  ; Show Stap 8 B
ANDNOT M_Show_Stap_9  ; Show Stap 9
ANDNOT M_Show_Stap_10  ; Show Stap 10
SET Com1_Show_Stap_4  ; Show Stap 4
RSET Com1_Stap_3  ; Show Stap 3
; rung 25
LD Com1_Show_Stap_4  ; Show Stap 4
AND COM2_STAP4  ; STAP 4 CYCLUS
OUT M_Show_Stap_4  ; Show Stap 4
; rung 26: Vertragingstijd t.b.v. de show Rotatie Eiland Als de Arm Boven is
LD Com1_Show_Stap_4  ; Show Stap 4
TIM 0115 D2939  ; EILAND TIJD BOVEN
; rung 27: (Show Stap 5) Start Arm Beweging Omlaag
LD>=S(327) D_PLC2_ENCODE1 +7000  ; GRADEN GETAL ENCODER 1
AND>=S(327) D_PLC2_ENCODE2 +7000  ; GRADEN GETAL ENCODER 2
AND T_EILAND_BOVEN  ; EILAND TIJD BOVEN
ANDNOT M_Show_Stap_0  ; Show Stap 0
ANDNOT M_Show_Stap_1  ; Show Stap 1
ANDNOT M_Show_Stap_2  ; Show Stap 2
ANDNOT M_Show_Stap_3  ; Show Stap 3
AND Com1_Show_Stap_4  ; Show Stap 4
ANDNOT M_Show_Stap_5  ; Show Stap 5
ANDNOT M_Show_Stap_6  ; Show Stap 6
ANDNOT M_Show_Stap_7  ; Show Stap 7
ANDNOT M_Show_Stap_8  ; Show Stap 8
ANDNOT Com1_Show_Stap_8A  ; Show Stap 8 A
ANDNOT Com1_Show_Stap_8B  ; Show Stap 8 B
ANDNOT M_Show_Stap_9  ; Show Stap 9
ANDNOT M_Show_Stap_10  ; Show Stap 10
SET Com1_Show_Stap_5  ; Show Stap 5
RSET Com1_Show_Stap_4  ; Show Stap 4
; rung 28
LD Com1_Show_Stap_5  ; Show Stap 5
AND Com2_Show_Stap_5  ; Show _Stap_5
OUT M_Show_Stap_5  ; Show Stap 5

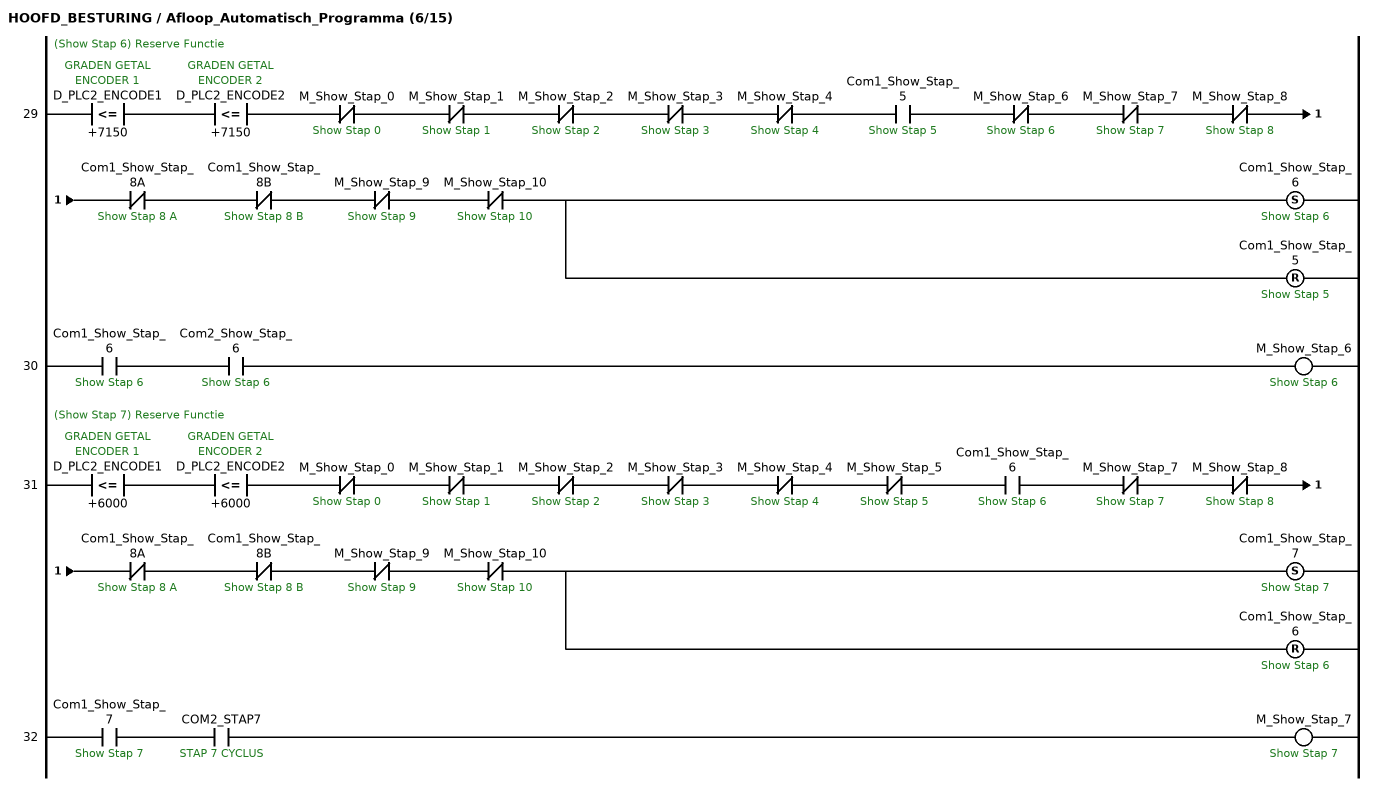
; rung 29: (Show Stap 6) Reserve Functie
LD<=S(317) D_PLC2_ENCODE1 +7150  ; GRADEN GETAL ENCODER 1
AND<=S(317) D_PLC2_ENCODE2 +7150  ; GRADEN GETAL ENCODER 2
ANDNOT M_Show_Stap_0  ; Show Stap 0
ANDNOT M_Show_Stap_1  ; Show Stap 1
ANDNOT M_Show_Stap_2  ; Show Stap 2
ANDNOT M_Show_Stap_3  ; Show Stap 3
ANDNOT M_Show_Stap_4  ; Show Stap 4
AND Com1_Show_Stap_5  ; Show Stap 5
ANDNOT M_Show_Stap_6  ; Show Stap 6
ANDNOT M_Show_Stap_7  ; Show Stap 7
ANDNOT M_Show_Stap_8  ; Show Stap 8
ANDNOT Com1_Show_Stap_8A  ; Show Stap 8 A
ANDNOT Com1_Show_Stap_8B  ; Show Stap 8 B
ANDNOT M_Show_Stap_9  ; Show Stap 9
ANDNOT M_Show_Stap_10  ; Show Stap 10
SET Com1_Show_Stap_6  ; Show Stap 6
RSET Com1_Show_Stap_5  ; Show Stap 5
; rung 30
LD Com1_Show_Stap_6  ; Show Stap 6
AND Com2_Show_Stap_6  ; Show Stap 6
OUT M_Show_Stap_6  ; Show Stap 6
; rung 31: (Show Stap 7) Reserve Functie
LD<=S(317) D_PLC2_ENCODE1 +6000  ; GRADEN GETAL ENCODER 1
AND<=S(317) D_PLC2_ENCODE2 +6000  ; GRADEN GETAL ENCODER 2
ANDNOT M_Show_Stap_0  ; Show Stap 0
ANDNOT M_Show_Stap_1  ; Show Stap 1
ANDNOT M_Show_Stap_2  ; Show Stap 2
ANDNOT M_Show_Stap_3  ; Show Stap 3
ANDNOT M_Show_Stap_4  ; Show Stap 4
ANDNOT M_Show_Stap_5  ; Show Stap 5
AND Com1_Show_Stap_6  ; Show Stap 6
ANDNOT M_Show_Stap_7  ; Show Stap 7
ANDNOT M_Show_Stap_8  ; Show Stap 8
ANDNOT Com1_Show_Stap_8A  ; Show Stap 8 A
ANDNOT Com1_Show_Stap_8B  ; Show Stap 8 B
ANDNOT M_Show_Stap_9  ; Show Stap 9
ANDNOT M_Show_Stap_10  ; Show Stap 10
SET Com1_Show_Stap_7  ; Show Stap 7
RSET Com1_Show_Stap_6  ; Show Stap 6
; rung 32
LD Com1_Show_Stap_7  ; Show Stap 7
AND COM2_STAP7  ; STAP 7 CYCLUS
OUT M_Show_Stap_7  ; Show Stap 7

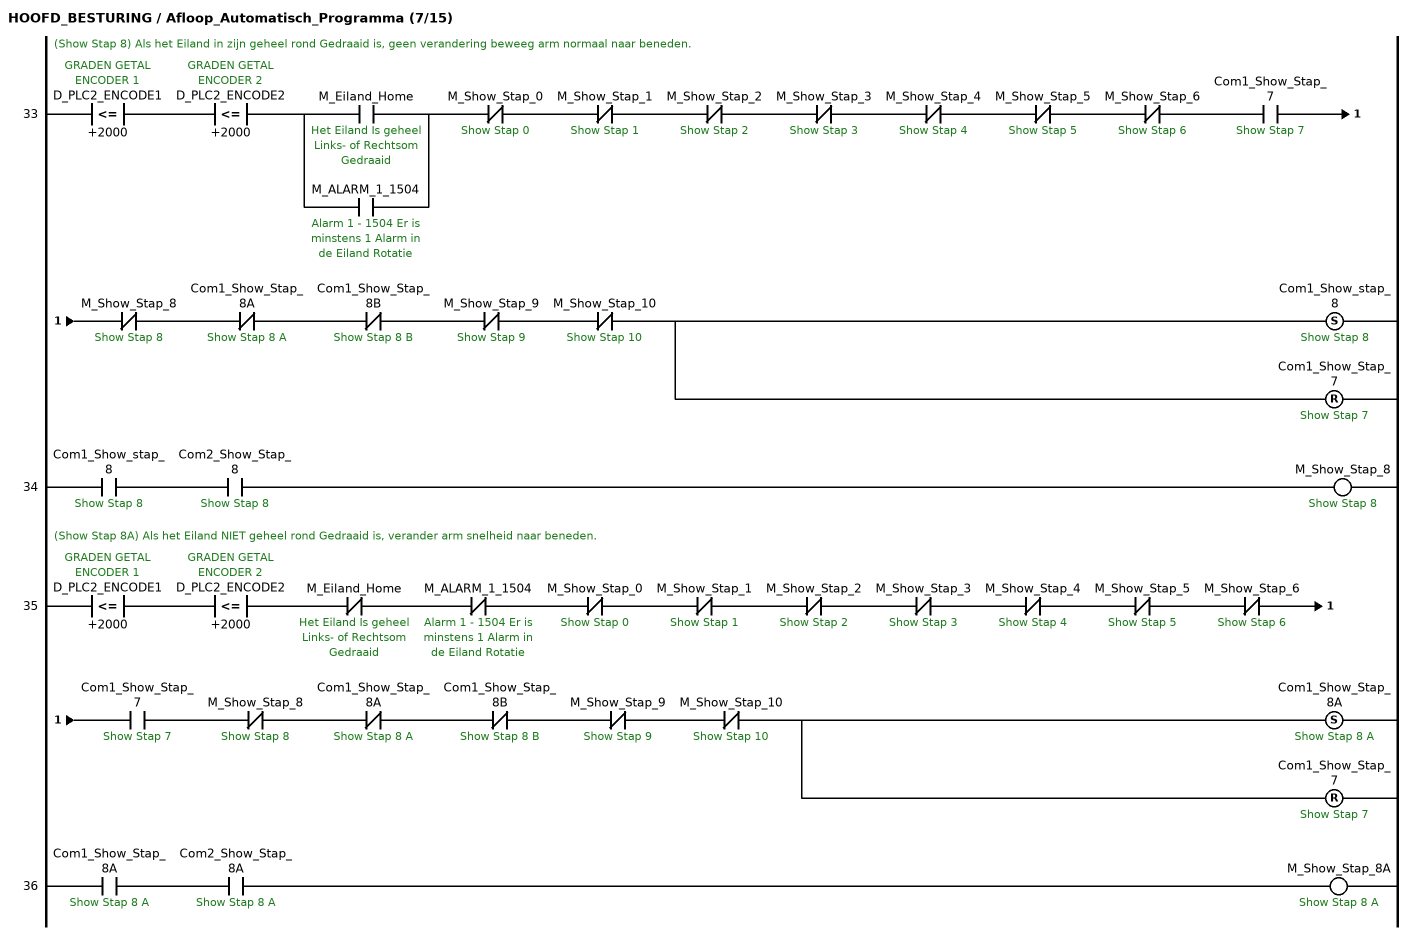
; rung 33: (Show Stap 8) Als het Eiland in zijn geheel rond Gedraaid is, geen verandering beweeg arm normaal naar beneden.
LD<=S(317) D_PLC2_ENCODE1 +2000  ; GRADEN GETAL ENCODER 1
AND<=S(317) D_PLC2_ENCODE2 +2000  ; GRADEN GETAL ENCODER 2
LD M_Eiland_Home  ; Het Eiland Is geheel Links- of Rechtsom Gedraaid
OR M_ALARM_1_1504  ; Alarm 1 - 1504 Er is minstens 1 Alarm in de Eiland Rotatie
ANDLD
ANDNOT M_Show_Stap_0  ; Show Stap 0
ANDNOT M_Show_Stap_1  ; Show Stap 1
ANDNOT M_Show_Stap_2  ; Show Stap 2
ANDNOT M_Show_Stap_3  ; Show Stap 3
ANDNOT M_Show_Stap_4  ; Show Stap 4
ANDNOT M_Show_Stap_5  ; Show Stap 5
ANDNOT M_Show_Stap_6  ; Show Stap 6
AND Com1_Show_Stap_7  ; Show Stap 7
ANDNOT M_Show_Stap_8  ; Show Stap 8
ANDNOT Com1_Show_Stap_8A  ; Show Stap 8 A
ANDNOT Com1_Show_Stap_8B  ; Show Stap 8 B
ANDNOT M_Show_Stap_9  ; Show Stap 9
ANDNOT M_Show_Stap_10  ; Show Stap 10
SET Com1_Show_stap_8  ; Show Stap 8
RSET Com1_Show_Stap_7  ; Show Stap 7
; rung 34
LD Com1_Show_stap_8  ; Show Stap 8
AND Com2_Show_Stap_8  ; Show Stap 8
OUT M_Show_Stap_8  ; Show Stap 8
; rung 35: (Show Stap 8A) Als het Eiland NIET geheel rond Gedraaid is, verander arm snelheid naar beneden.
LD<=S(317) D_PLC2_ENCODE1 +2000  ; GRADEN GETAL ENCODER 1
AND<=S(317) D_PLC2_ENCODE2 +2000  ; GRADEN GETAL ENCODER 2
ANDNOT M_Eiland_Home  ; Het Eiland Is geheel Links- of Rechtsom Gedraaid
ANDNOT M_ALARM_1_1504  ; Alarm 1 - 1504 Er is minstens 1 Alarm in de Eiland Rotatie
ANDNOT M_Show_Stap_0  ; Show Stap 0
ANDNOT M_Show_Stap_1  ; Show Stap 1
ANDNOT M_Show_Stap_2  ; Show Stap 2
ANDNOT M_Show_Stap_3  ; Show Stap 3
ANDNOT M_Show_Stap_4  ; Show Stap 4
ANDNOT M_Show_Stap_5  ; Show Stap 5
ANDNOT M_Show_Stap_6  ; Show Stap 6
AND Com1_Show_Stap_7  ; Show Stap 7
ANDNOT M_Show_Stap_8  ; Show Stap 8
ANDNOT Com1_Show_Stap_8A  ; Show Stap 8 A
ANDNOT Com1_Show_Stap_8B  ; Show Stap 8 B
ANDNOT M_Show_Stap_9  ; Show Stap 9
ANDNOT M_Show_Stap_10  ; Show Stap 10
SET Com1_Show_Stap_8A  ; Show Stap 8 A
RSET Com1_Show_Stap_7  ; Show Stap 7
; rung 36
LD Com1_Show_Stap_8A  ; Show Stap 8 A
AND Com2_Show_Stap_8A  ; Show Stap 8 A
OUT M_Show_Stap_8A  ; Show Stap 8 A

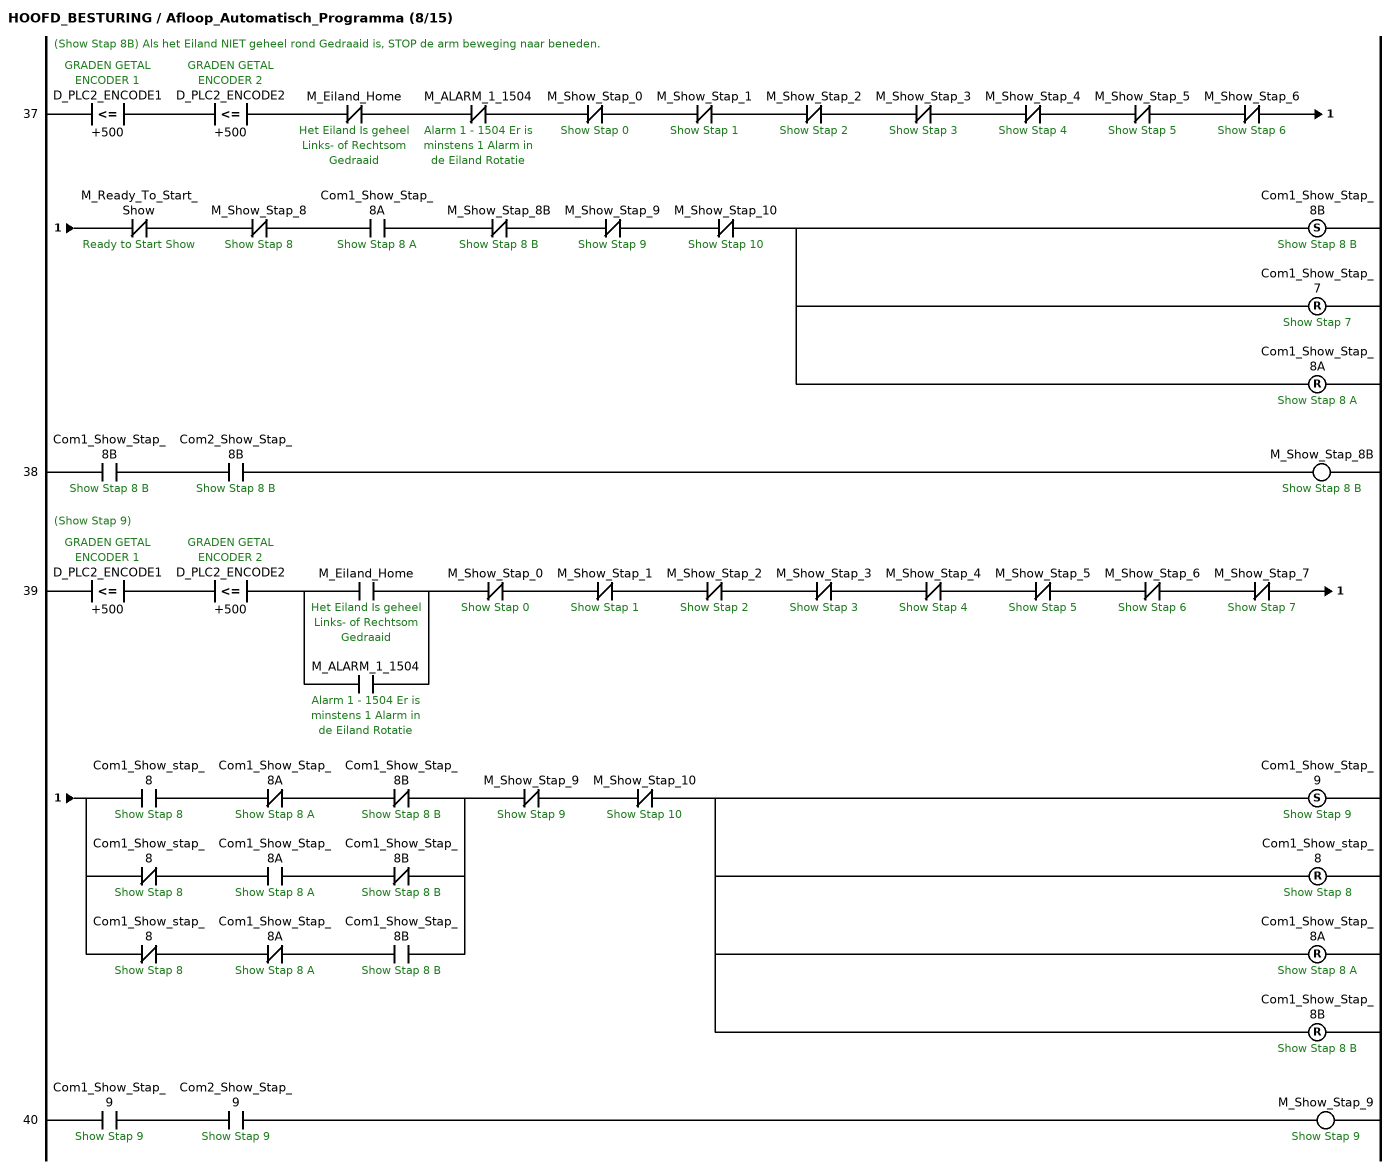
; rung 37: (Show Stap 8B) Als het Eiland NIET geheel rond Gedraaid is, STOP de arm beweging naar beneden.
LD<=S(317) D_PLC2_ENCODE1 +500  ; GRADEN GETAL ENCODER 1
AND<=S(317) D_PLC2_ENCODE2 +500  ; GRADEN GETAL ENCODER 2
ANDNOT M_Eiland_Home  ; Het Eiland Is geheel Links- of Rechtsom Gedraaid
ANDNOT M_ALARM_1_1504  ; Alarm 1 - 1504 Er is minstens 1 Alarm in de Eiland Rotatie
ANDNOT M_Show_Stap_0  ; Show Stap 0
ANDNOT M_Show_Stap_1  ; Show Stap 1
ANDNOT M_Show_Stap_2  ; Show Stap 2
ANDNOT M_Show_Stap_3  ; Show Stap 3
ANDNOT M_Show_Stap_4  ; Show Stap 4
ANDNOT M_Show_Stap_5  ; Show Stap 5
ANDNOT M_Show_Stap_6  ; Show Stap 6
ANDNOT M_Ready_To_Start_Show  ; Ready to Start Show
ANDNOT M_Show_Stap_8  ; Show Stap 8
AND Com1_Show_Stap_8A  ; Show Stap 8 A
ANDNOT M_Show_Stap_8B  ; Show Stap 8 B
ANDNOT M_Show_Stap_9  ; Show Stap 9
ANDNOT M_Show_Stap_10  ; Show Stap 10
SET Com1_Show_Stap_8B  ; Show Stap 8 B
RSET Com1_Show_Stap_7  ; Show Stap 7
RSET Com1_Show_Stap_8A  ; Show Stap 8 A
; rung 38
LD Com1_Show_Stap_8B  ; Show Stap 8 B
AND Com2_Show_Stap_8B  ; Show Stap 8 B
OUT M_Show_Stap_8B  ; Show Stap 8 B
; rung 39: (Show Stap 9)
LD<=S(317) D_PLC2_ENCODE1 +500  ; GRADEN GETAL ENCODER 1
AND<=S(317) D_PLC2_ENCODE2 +500  ; GRADEN GETAL ENCODER 2
LD M_Eiland_Home  ; Het Eiland Is geheel Links- of Rechtsom Gedraaid
OR M_ALARM_1_1504  ; Alarm 1 - 1504 Er is minstens 1 Alarm in de Eiland Rotatie
ANDLD
ANDNOT M_Show_Stap_0  ; Show Stap 0
ANDNOT M_Show_Stap_1  ; Show Stap 1
ANDNOT M_Show_Stap_2  ; Show Stap 2
ANDNOT M_Show_Stap_3  ; Show Stap 3
ANDNOT M_Show_Stap_4  ; Show Stap 4
ANDNOT M_Show_Stap_5  ; Show Stap 5
ANDNOT M_Show_Stap_6  ; Show Stap 6
ANDNOT M_Show_Stap_7  ; Show Stap 7
LD Com1_Show_stap_8  ; Show Stap 8
ANDNOT Com1_Show_Stap_8A  ; Show Stap 8 A
ANDNOT Com1_Show_Stap_8B  ; Show Stap 8 B
LDNOT Com1_Show_stap_8  ; Show Stap 8
AND Com1_Show_Stap_8A  ; Show Stap 8 A
ANDNOT Com1_Show_Stap_8B  ; Show Stap 8 B
ORLD
LDNOT Com1_Show_stap_8  ; Show Stap 8
ANDNOT Com1_Show_Stap_8A  ; Show Stap 8 A
AND Com1_Show_Stap_8B  ; Show Stap 8 B
ORLD
ANDLD
ANDNOT M_Show_Stap_9  ; Show Stap 9
ANDNOT M_Show_Stap_10  ; Show Stap 10
SET Com1_Show_Stap_9  ; Show Stap 9
RSET Com1_Show_stap_8  ; Show Stap 8
RSET Com1_Show_Stap_8A  ; Show Stap 8 A
RSET Com1_Show_Stap_8B  ; Show Stap 8 B
; rung 40
LD Com1_Show_Stap_9  ; Show Stap 9
AND Com2_Show_Stap_9  ; Show Stap 9
OUT M_Show_Stap_9  ; Show Stap 9

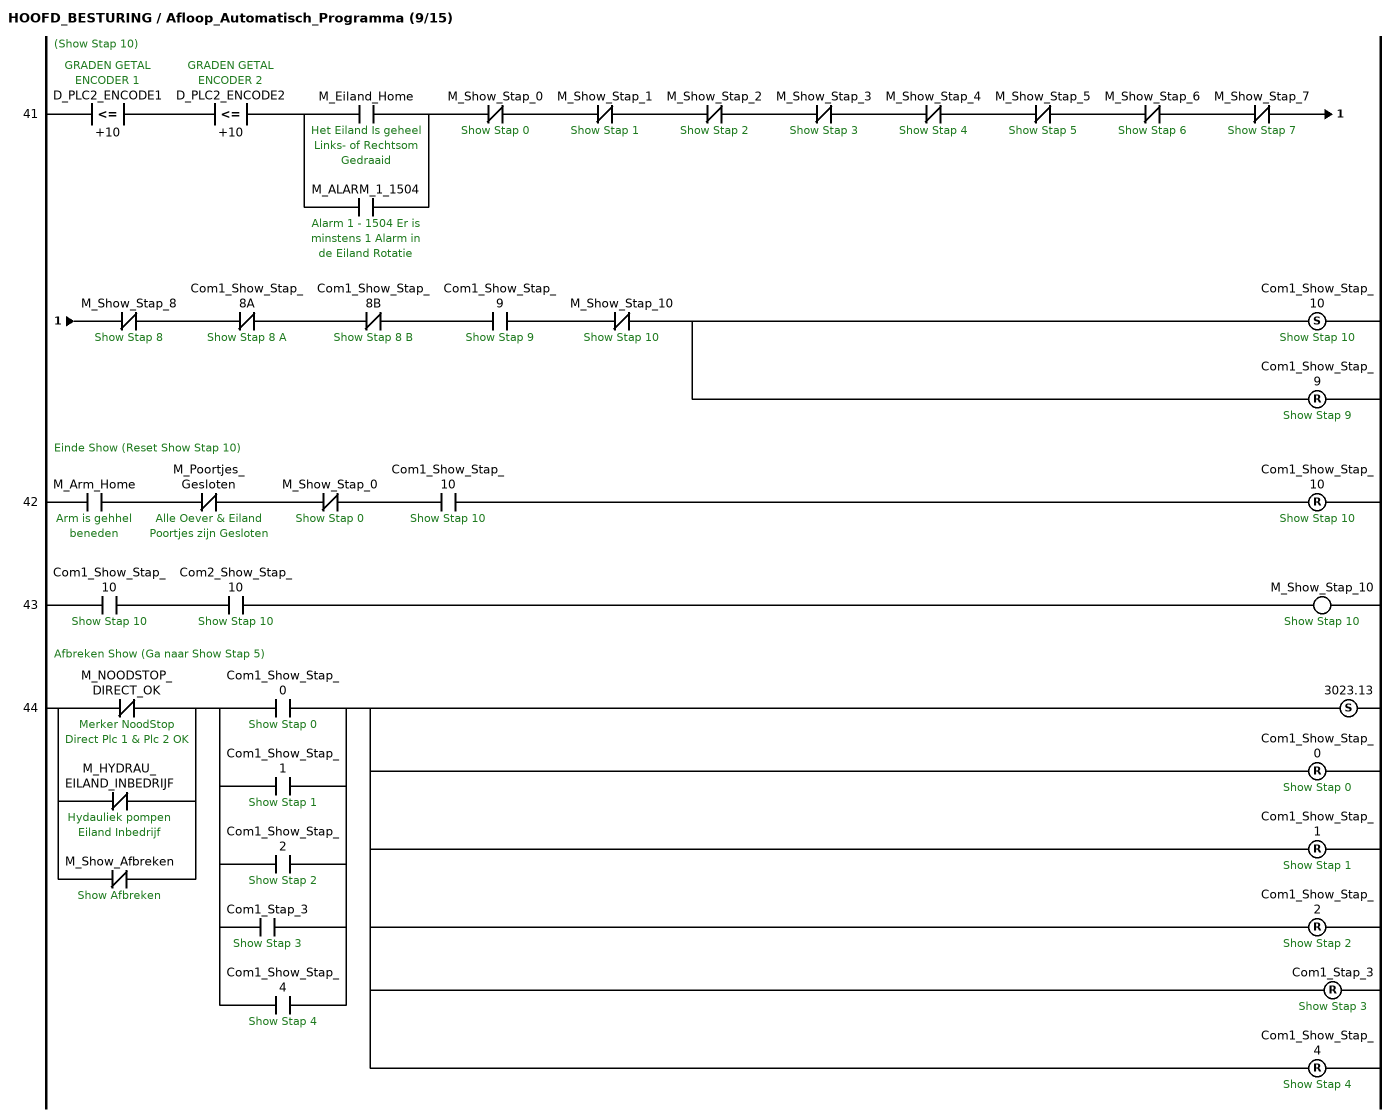
; rung 41: (Show Stap 10)
LD<=S(317) D_PLC2_ENCODE1 +10  ; GRADEN GETAL ENCODER 1
AND<=S(317) D_PLC2_ENCODE2 +10  ; GRADEN GETAL ENCODER 2
LD M_Eiland_Home  ; Het Eiland Is geheel Links- of Rechtsom Gedraaid
OR M_ALARM_1_1504  ; Alarm 1 - 1504 Er is minstens 1 Alarm in de Eiland Rotatie
ANDLD
ANDNOT M_Show_Stap_0  ; Show Stap 0
ANDNOT M_Show_Stap_1  ; Show Stap 1
ANDNOT M_Show_Stap_2  ; Show Stap 2
ANDNOT M_Show_Stap_3  ; Show Stap 3
ANDNOT M_Show_Stap_4  ; Show Stap 4
ANDNOT M_Show_Stap_5  ; Show Stap 5
ANDNOT M_Show_Stap_6  ; Show Stap 6
ANDNOT M_Show_Stap_7  ; Show Stap 7
ANDNOT M_Show_Stap_8  ; Show Stap 8
ANDNOT Com1_Show_Stap_8A  ; Show Stap 8 A
ANDNOT Com1_Show_Stap_8B  ; Show Stap 8 B
AND Com1_Show_Stap_9  ; Show Stap 9
ANDNOT M_Show_Stap_10  ; Show Stap 10
SET Com1_Show_Stap_10  ; Show Stap 10
RSET Com1_Show_Stap_9  ; Show Stap 9
; rung 42: Einde Show (Reset Show Stap 10)
LD M_Arm_Home  ; Arm is gehhel beneden
ANDNOT M_Poortjes_Gesloten  ; Alle Oever & Eiland Poortjes zijn Gesloten
ANDNOT M_Show_Stap_0  ; Show Stap 0
AND Com1_Show_Stap_10  ; Show Stap 10
RSET Com1_Show_Stap_10  ; Show Stap 10
; rung 43
LD Com1_Show_Stap_10  ; Show Stap 10
AND Com2_Show_Stap_10  ; Show Stap 10
OUT M_Show_Stap_10  ; Show Stap 10
; rung 44: Afbreken Show (Ga naar Show Stap 5)
LDNOT M_NOODSTOP_DIRECT_OK  ; Merker NoodStop Direct Plc 1 & Plc 2 OK
ORNOT M_HYDRAU_EILAND_INBEDRIJF  ; Hydauliek pompen Eiland Inbedrijf
ORNOT M_Show_Afbreken  ; Show Afbreken
LD Com1_Show_Stap_0  ; Show Stap 0
OR Com1_Show_Stap_1  ; Show Stap 1
OR Com1_Show_Stap_2  ; Show Stap 2
OR Com1_Stap_3  ; Show Stap 3
OR Com1_Show_Stap_4  ; Show Stap 4
ANDLD
SET 3023.13
RSET Com1_Show_Stap_0  ; Show Stap 0
RSET Com1_Show_Stap_1  ; Show Stap 1
RSET Com1_Show_Stap_2  ; Show Stap 2
RSET Com1_Stap_3  ; Show Stap 3
RSET Com1_Show_Stap_4  ; Show Stap 4

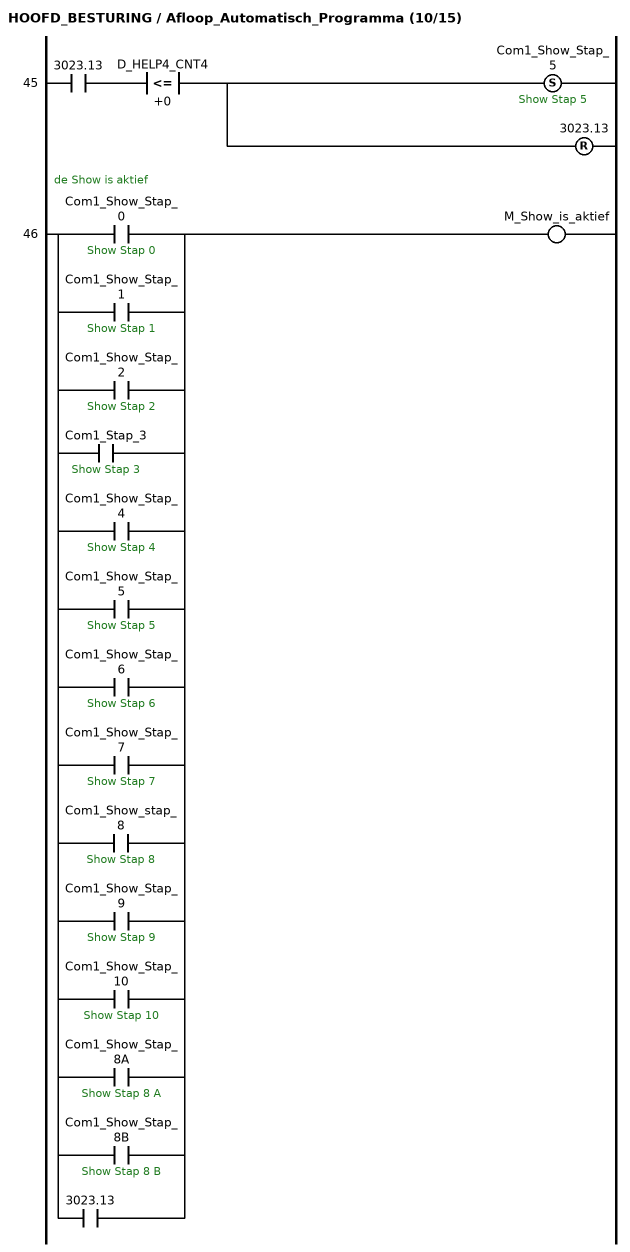
; rung 45
LD 3023.13
AND<=S(317) D_HELP4_CNT4 +0
SET Com1_Show_Stap_5  ; Show Stap 5
RSET 3023.13
; rung 46: de Show is aktief
LD Com1_Show_Stap_0  ; Show Stap 0
OR Com1_Show_Stap_1  ; Show Stap 1
OR Com1_Show_Stap_2  ; Show Stap 2
OR Com1_Stap_3  ; Show Stap 3
OR Com1_Show_Stap_4  ; Show Stap 4
OR Com1_Show_Stap_5  ; Show Stap 5
OR Com1_Show_Stap_6  ; Show Stap 6
OR Com1_Show_Stap_7  ; Show Stap 7
OR Com1_Show_stap_8  ; Show Stap 8
OR Com1_Show_Stap_9  ; Show Stap 9
OR Com1_Show_Stap_10  ; Show Stap 10
OR Com1_Show_Stap_8A  ; Show Stap 8 A
OR Com1_Show_Stap_8B  ; Show Stap 8 B
OR 3023.13
OUT M_Show_is_aktief

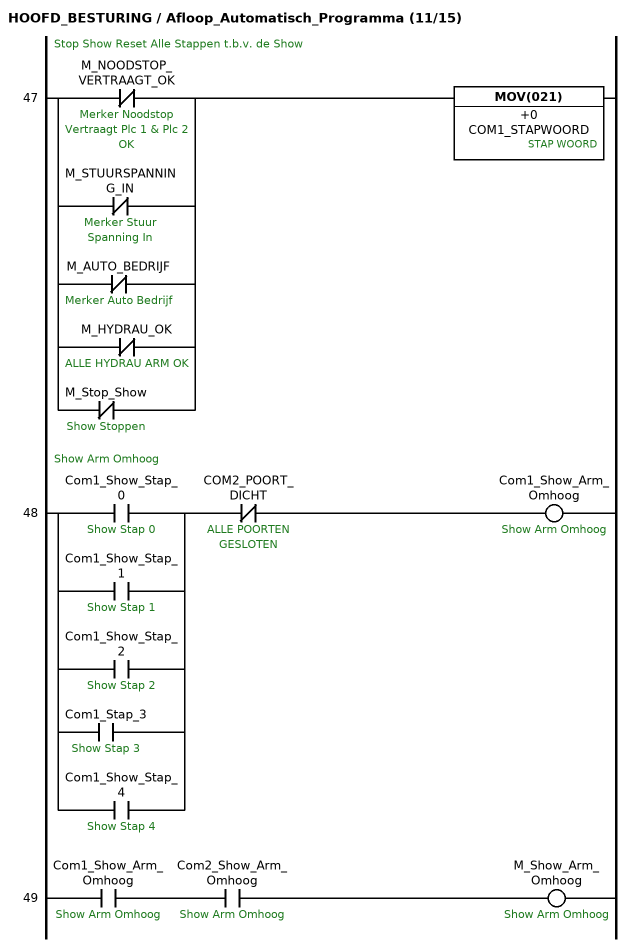
; rung 47: Stop Show Reset Alle Stappen t.b.v. de Show
LDNOT M_NOODSTOP_VERTRAAGT_OK  ; Merker Noodstop Vertraagt Plc 1 & Plc 2 OK
ORNOT M_STUURSPANNING_IN  ; Merker Stuur Spanning In
ORNOT M_AUTO_BEDRIJF  ; Merker Auto Bedrijf
ORNOT M_HYDRAU_OK  ; ALLE HYDRAU ARM OK
ORNOT M_Stop_Show  ; Show Stoppen
MOV(021) +0 COM1_STAPWOORD  ; STAP WOORD
; rung 48: Show Arm Omhoog
LD Com1_Show_Stap_0  ; Show Stap 0
OR Com1_Show_Stap_1  ; Show Stap 1
OR Com1_Show_Stap_2  ; Show Stap 2
OR Com1_Stap_3  ; Show Stap 3
OR Com1_Show_Stap_4  ; Show Stap 4
ANDNOT COM2_POORT_DICHT  ; ALLE POORTEN GESLOTEN
OUT Com1_Show_Arm_Omhoog  ; Show Arm Omhoog
; rung 49
LD Com1_Show_Arm_Omhoog  ; Show Arm Omhoog
AND Com2_Show_Arm_Omhoog  ; Show Arm Omhoog
OUT M_Show_Arm_Omhoog  ; Show Arm Omhoog

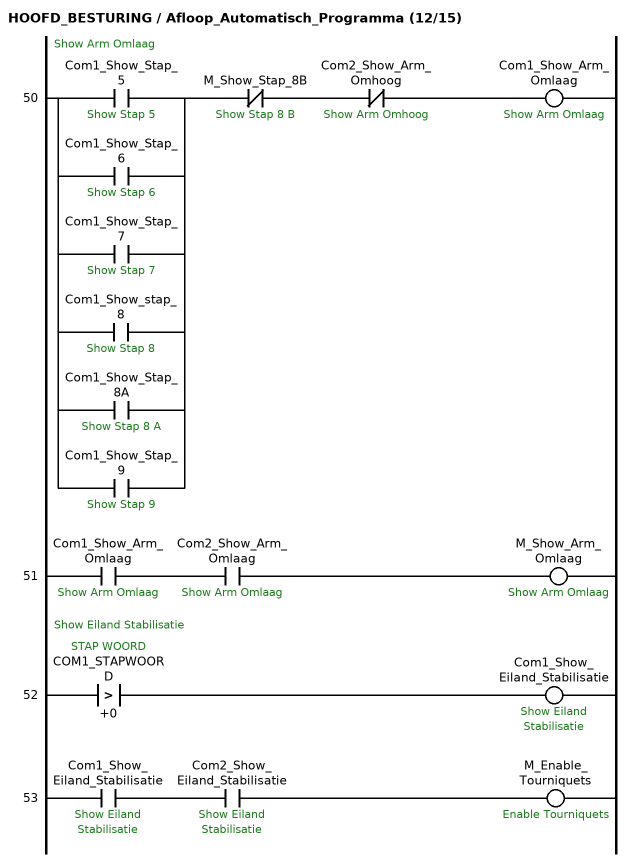
; rung 50: Show Arm Omlaag
LD Com1_Show_Stap_5  ; Show Stap 5
OR Com1_Show_Stap_6  ; Show Stap 6
OR Com1_Show_Stap_7  ; Show Stap 7
OR Com1_Show_stap_8  ; Show Stap 8
OR Com1_Show_Stap_8A  ; Show Stap 8 A
OR Com1_Show_Stap_9  ; Show Stap 9
ANDNOT M_Show_Stap_8B  ; Show Stap 8 B
ANDNOT Com2_Show_Arm_Omhoog  ; Show Arm Omhoog
OUT Com1_Show_Arm_Omlaag  ; Show Arm Omlaag
; rung 51
LD Com1_Show_Arm_Omlaag  ; Show Arm Omlaag
AND Com2_Show_Arm_Omlaag  ; Show Arm Omlaag
OUT M_Show_Arm_Omlaag  ; Show Arm Omlaag
; rung 52: Show Eiland Stabilisatie
LD>S(322) COM1_STAPWOORD +0  ; STAP WOORD
OUT Com1_Show_Eiland_Stabilisatie  ; Show Eiland Stabilisatie
; rung 53
LD Com1_Show_Eiland_Stabilisatie  ; Show Eiland Stabilisatie
AND Com2_Show_Eiland_Stabilisatie  ; Show Eiland Stabilisatie
OUT M_Enable_Tourniquets  ; Enable Tourniquets

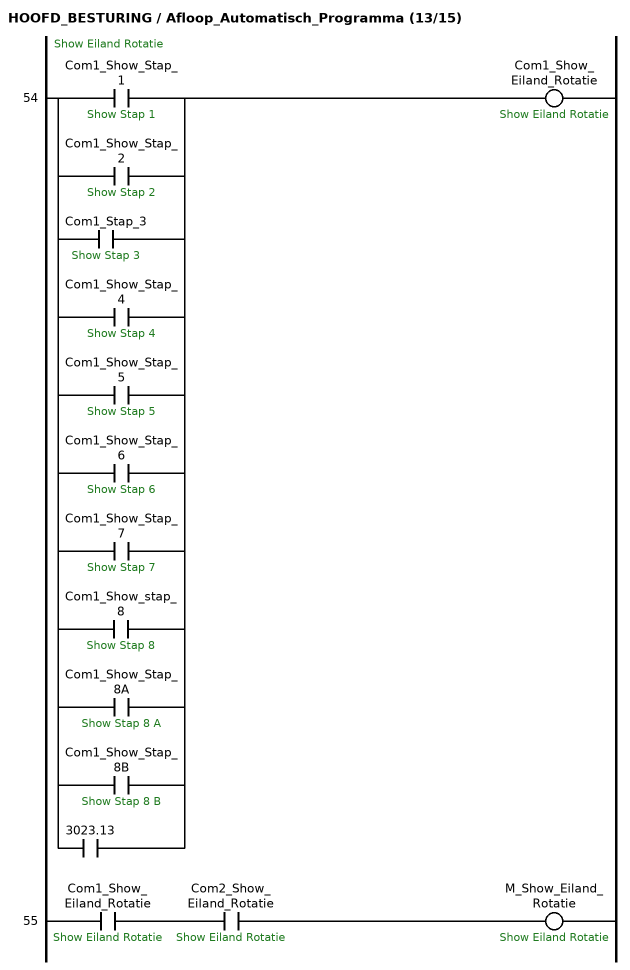
; rung 54: Show Eiland Rotatie
LD Com1_Show_Stap_1  ; Show Stap 1
OR Com1_Show_Stap_2  ; Show Stap 2
OR Com1_Stap_3  ; Show Stap 3
OR Com1_Show_Stap_4  ; Show Stap 4
OR Com1_Show_Stap_5  ; Show Stap 5
OR Com1_Show_Stap_6  ; Show Stap 6
OR Com1_Show_Stap_7  ; Show Stap 7
OR Com1_Show_stap_8  ; Show Stap 8
OR Com1_Show_Stap_8A  ; Show Stap 8 A
OR Com1_Show_Stap_8B  ; Show Stap 8 B
OR 3023.13
OUT Com1_Show_Eiland_Rotatie  ; Show Eiland Rotatie
; rung 55
LD Com1_Show_Eiland_Rotatie  ; Show Eiland Rotatie
AND Com2_Show_Eiland_Rotatie  ; Show Eiland Rotatie
OUT M_Show_Eiland_Rotatie  ; Show Eiland Rotatie

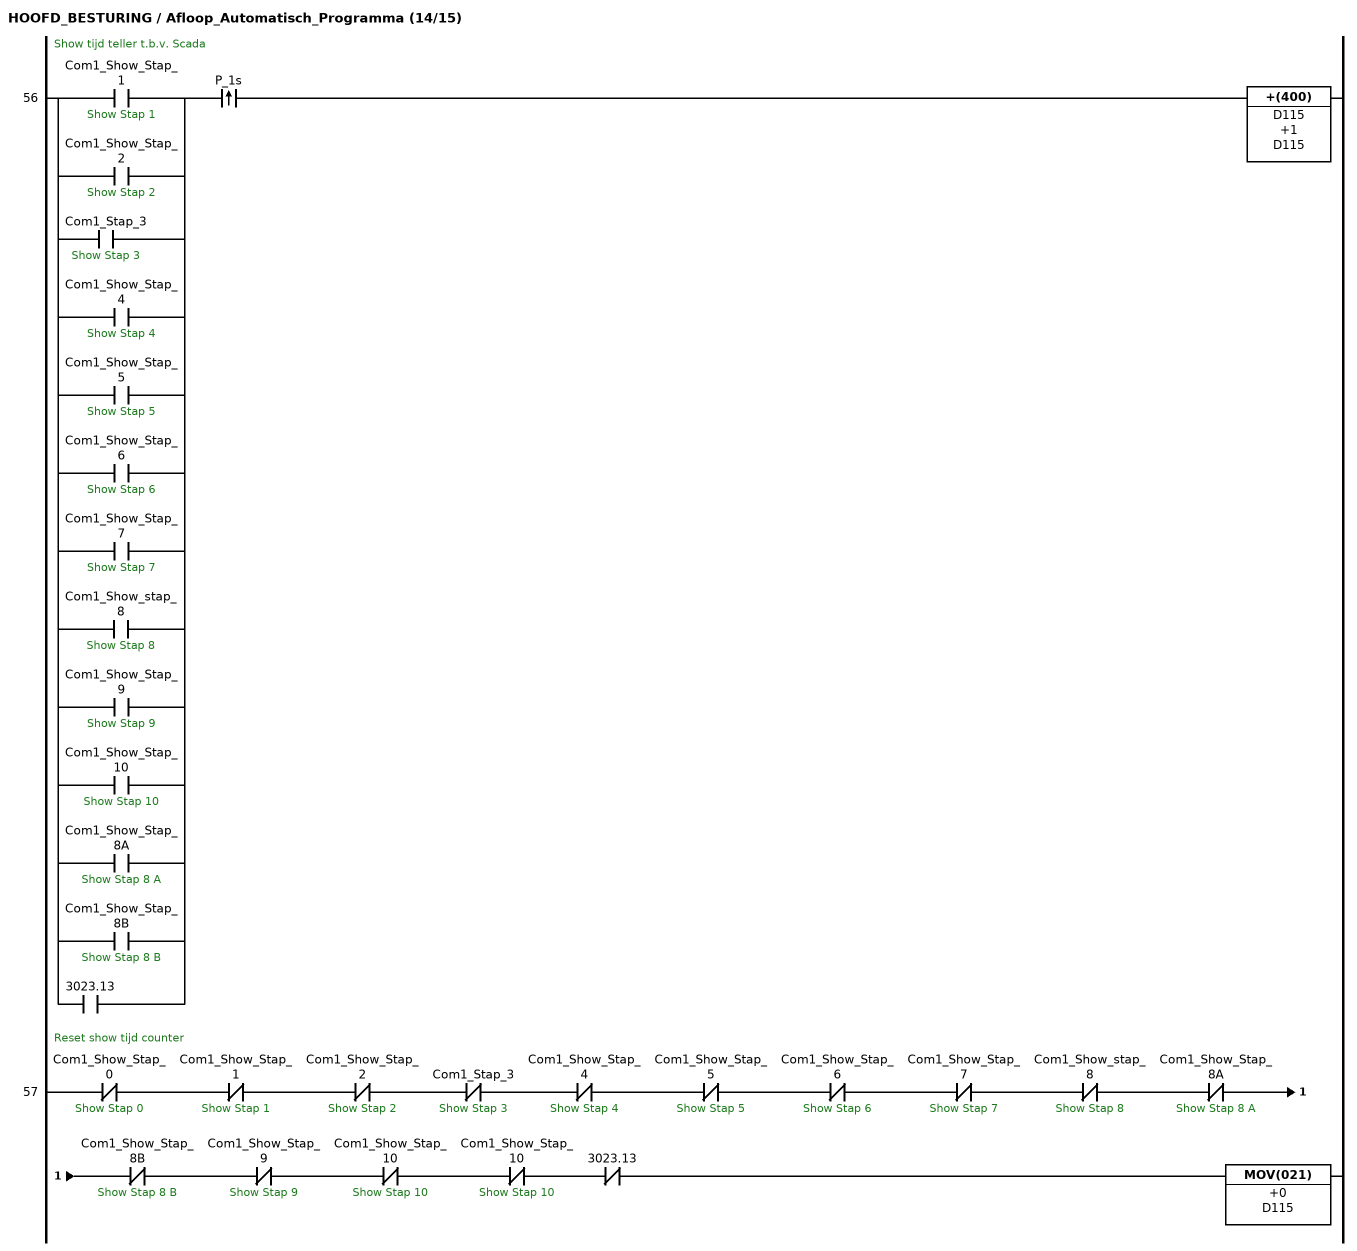
; rung 56: Show tijd teller t.b.v. Scada
LD Com1_Show_Stap_1  ; Show Stap 1
OR Com1_Show_Stap_2  ; Show Stap 2
OR Com1_Stap_3  ; Show Stap 3
OR Com1_Show_Stap_4  ; Show Stap 4
OR Com1_Show_Stap_5  ; Show Stap 5
OR Com1_Show_Stap_6  ; Show Stap 6
OR Com1_Show_Stap_7  ; Show Stap 7
OR Com1_Show_stap_8  ; Show Stap 8
OR Com1_Show_Stap_9  ; Show Stap 9
OR Com1_Show_Stap_10  ; Show Stap 10
OR Com1_Show_Stap_8A  ; Show Stap 8 A
OR Com1_Show_Stap_8B  ; Show Stap 8 B
OR 3023.13
@AND P_1s
+(400) D115 +1 D115
; rung 57: Reset show tijd counter
LDNOT Com1_Show_Stap_0  ; Show Stap 0
ANDNOT Com1_Show_Stap_1  ; Show Stap 1
ANDNOT Com1_Show_Stap_2  ; Show Stap 2
ANDNOT Com1_Stap_3  ; Show Stap 3
ANDNOT Com1_Show_Stap_4  ; Show Stap 4
ANDNOT Com1_Show_Stap_5  ; Show Stap 5
ANDNOT Com1_Show_Stap_6  ; Show Stap 6
ANDNOT Com1_Show_Stap_7  ; Show Stap 7
ANDNOT Com1_Show_stap_8  ; Show Stap 8
ANDNOT Com1_Show_Stap_8A  ; Show Stap 8 A
ANDNOT Com1_Show_Stap_8B  ; Show Stap 8 B
ANDNOT Com1_Show_Stap_9  ; Show Stap 9
ANDNOT Com1_Show_Stap_10  ; Show Stap 10
ANDNOT Com1_Show_Stap_10  ; Show Stap 10
ANDNOT 3023.13
MOV(021) +0 D115

